      U(    ;
      U     "G271M".A_3125_MXZ01MA.Ma.StStartedFwd; // min one fan must run
      O     DB371.DBX 1445.2; // min one fan must run
      )     ;
      UN    "MAL1S032Par".Par.FlagProcess.Inf08; // Schritt halten
      UN    "G269M".A_3191_BTE07.OutOverflow; //LUFTTEMPERATUR ÜBER DER HORDE
      UN    "G269M".A_3191_BTE07.OutFaultAI; //LUFTTEMPERATUR ÜBER DER HORDE
      UN    "G269M".A_3191_BTE01.OutOverflow; //LUFTTEMPERATUR UNTER DER HORDE
      UN    "G269M".A_3191_BTE01.OutFaultAI; //LUFTTEMPERATUR UNTER DER HORDE
      SPBN  NoTi; // count steptime only when fan running and sensor alive
//JV161209      L     "MAL1S032Par".Par.ProcessValue.StepTimeAct    // in ms
//JV161209      L     #tmpCyclusTime
//JV161209      +D
//JV161209      T     "MAL1S032Par".Par.ProcessValue.StepTimeAct    // in ms
//--Create actual Timeinterval for counting steptime new JV151209 ===>

      CALL "SIEMENS_READ_CLK" (
           RET_VAL                  := MW   200,
           CDT                      := "MAL1S032Par".Par.ProcessValue.ActualTime);

      U     "MAL1S032Par".Par.FlagProcess.Inf04; // Zeitauswertung aktiv
      SPB   diff;
      CALL "SIEMENS_READ_CLK" (
           RET_VAL                  := MW   200,
           CDT                      := "MAL1S032Par".Par.ProcessValue.ActualTimePreviousScan);// Start-Zeit CPU-Clock aktuelle Auswertung
      SET   ;
      S     "MAL1S032Par".Par.FlagProcess.Inf04; // Zeitauswertung aktiv

diff: NOP   0;

      CALL "SB_DT_DT" (
           DT1                      := "MAL1S032Par".Par.ProcessValue.ActualTime,// momentane Zeit CPU-Clock
           DT2                      := "MAL1S032Par".Par.ProcessValue.ActualTimePreviousScan,// Start-Zeit CPU-Clock aktuelle Auswertung
           RET_VAL                  := "MAL1S032Par".Par.ProcessValue.Afeesttijd);// Zeitdifferenz in ms


      L     "MAL1S032Par".Par.ProcessValue.Afeesttijd; // Zeitdifferenz in ms
      L     L#10000; // 10sec
      >=D   ;
      R     "MAL1S032Par".Par.FlagProcess.Inf04; // Zeitauswertung aktiv
      FP    "MAL1S032Par".Par.FlagProcess.Inf05;
      SPBN  NoST;
      L     "MAL1S032Par".Par.ProcessValue.Afeesttijd; // Zeitdifferenz in ms
      SPM   Korr; //JV161209 Da hat wer an der Uhr gedreht.....
      L     L#10150; // 10sec + 150ms  als Maximalüberwachung
      >D    ; //JV161209 Da hat wer an der Uhr gedreht.....
      SPBN  AlOK;
Korr: NOP   0;
      L     L#10000; // 10sec als Grundwert, wenn die Zeit verstellt wurde
      T     "MAL1S032Par".Par.ProcessValue.Afeesttijd; // Zeitdifferenz in ms
AlOK: NOP   0;
      L     "MAL1S032Par".Par.ProcessValue.Afeesttijd; // Zeitdifferenz in ms
      L     "ASW_GraphicData".General.CycleTime[1].Actual; // aktuelle Zykluszeit als Korrektur
      +D    ;
      L     "MAL1S032Par".Par.ProcessValue.StepTimeAct; // in ms
      +D    ;
      T     "MAL1S032Par".Par.ProcessValue.StepTimeAct; // in ms
NoST: NOP   0;
//--Create actual Timeinterval for counting steptime new JV151209 <===

      SPA   OKTi; //JV161209
NoTi: NOP   0;
      SET   ; //JV161209 ===>
      R     "MAL1S032Par".Par.FlagProcess.Inf04; // Zeitauswertung aktiv
//JV161209 <===
OKTi: NOP   0; //JV161209
      L     "MAL1S032Par".Par.ProcessValue.StepTimeAct; // in ms
      L     L#86400000; // ms/d
      MOD   ;
      L     L#3600000; // ms/h
      /D    ;
      T     "MAL1S032Par".ActTimeStepProcess.SteptimeActHour; // Steptime in h

      L     "MAL1S032Par".Par.ProcessValue.StepTimeAct;
      L     L#3600000; // ms/h
      MOD   ;
      L     L#60000; // ms/min
      /D    ;
      T     "MAL1S032Par".ActTimeStepProcess.SteptimeActMin; // Steptime in min

      L     "MAL1S032Par".Par.ProcessValue.StepTimeAct;
      L     L#60000; // ms/min
      /D    ;
      T     "MAL1S032Par".ActTimeStepProcess.SteptimeActMinOverall; // Steptime in min overall

//
// Next Step
//
//   Switch over to next step under conditions:
//   or Maximal steptime
//   or Minimal steptime
//           and
//               or no setpoint delta temp
//               or atual value delta temp is ge setpoint deltatemp
//                   and sensor is ok
//           and
// /              or no setpoint max temp above floor
//              or atual value max temp above floor is ge setpoint max temp above floor
//                  and sensor is ok
// 1 Kriterium
      U(    ;
      L     "MAL1S032Par".ActTimeStepProcess.SteptimeActMinOverall; // Steptime in min overall
      L     "MAL1S032Par".StepAct.StepTime_Max; // Target steptime actual step
      >=I   ;
      )     ;
      O(    ;
// 2 Kriterium
      O(    ;
      U(    ;
      L     "MAL1S032Par".StepAct.DeltaTempSwitchpointStep;
      L     0;
//JV230310      >=D
      >D    ; //JV230310
      )     ;
// condition, if analogue input is not damaaged   //
      UN    "G269M".A_3191_BTE07.OutOverflow; //AIR TEMPERATURE ABOVE FLOOR
      UN    "G269M".A_3191_BTE07.OutFaultAI; //AIR TEMPERATURE ABOVE FLOOR
      UN    "G269M".A_3191_BTE01.OutOverflow; //AIR TEMPERATURE BELOW FLOOR
      UN    "G269M".A_3191_BTE01.OutFaultAI; //AIR TEMPERATURE BELOW FLOOR
      U(    ;
      L     "G269M".A_3191_BTE01.OutValueUnits; // act value temperature below floor
      L     "G269M".A_3191_BTE07.OutValueUnits; // act value temperature above floor
      -D    ; // delta temp actual
      L     L#10;
      /D    ;
      L     "MAL1S032Par".StepAct.DeltaTempSwitchpointStep;
      <D    ;
      )     ;
      )     ;
// 3 Kriterium
      O(    ;
      U(    ;
      L     "MAL1S032Par".StepAct.MaxTempAboveFloorStep;
      L     L#0; // 0,0°C is illegally switchpoint for max. temperature
      >D    ;
      )     ;
// condition, if analogue input is not damaaged   // MW R2.1
      UN    "G269M".A_3191_BTE01.OutOverflow; //AIR TEMPERATURE BELOW FLOOR
      UN    "G269M".A_3191_BTE01.OutFaultAI; //AIR TEMPERATURE BELOW FLOOR
      U(    ;
      L     "G269M".A_3191_BTE07.OutValueUnits; // act value temperature above floor
      L     L#10;
      /D    ;
      L     "MAL1S032Par".StepAct.MaxTempAboveFloorStep;
      >=D   ;
      )     ;
      )     ;
// 4 Kriterium
// and min. time
      U(    ;
      L     "MAL1S032Par".ActTimeStepProcess.SteptimeActMinOverall; // Steptime in min overall
      L     "MAL1S032Par".StepAct.StepTime_Min; // Target steptime actual step
      >=I   ;
      )     ;
      )     ;
// and not cooling                                // UK 22.01.07
      UN    "MAL1S032Par".Par.FlagProcess.Cooling_Activ;
// 5 Kriterium
      O(    ;
      U     "MAL1S032Par".Par.FlagProcess.Cooling_Activ;
      U(    ;
      L     "G269M".A_3191_BTE07.OutValueUnits; // act value temperature above floor
      L     L#10;
      /D    ;
      L     "MAL1S032Par".StepAct.TemperaturAboveFloor;
      <=D   ;
      )     ;
      O(    ;
      L     "MAL1S032Par".Par.ParIntMachine.ActualStep;
//JV210710      L     25                          // max. 24 Schritte
      L     27; // max. 26 Schritte   //JV210710
      >=I   ;
      )     ;
      )     ;
// and min. time
      U(    ;
      L     "MAL1S032Par".ActTimeStepProcess.SteptimeActMinOverall; // Steptime in min overall
      L     "MAL1S032Par".StepAct.StepTime_Min; // Target steptime actual step
      >=I   ;
      )     ;
      SPBN  E606;
// send average step data to PIC
      SET   ;
      S     "MAL1S032StepValues".SendData; // send average step data to PIC
// Next step
      L     "MAL1S032Par".Par.ParIntMachine.ActualStep;
      L     "MAL1S032Par".RecipeHeader.NumberOfSteps;
      >I    ;
      SPB   Pedk; // Last step is finished
//BRT20100901 ====> Schritt halten
      U     "MAL1S032Par".Par.FlagProcess.Inf08; // Schritt halten
      SPB   E606;
//BRT20100901 <====
//
      L     "MAL1S032Par".Par.ParIntMachine.ActualStep;
      L     1;
      +I    ;
      T     "MAL1S032Par".Par.ParIntMachine.ActualStep;
      L     0;
      T     "MAL1S032Par".ActTimeStepProcess.SteptimeActMinOverall; // Steptime in min Overall
      SPA   E606;
Pedk: NOP   0; // Process has finished
      SET   ;
      R     "MAL1S032Par".Par.FlagProcess.ProcessActive;
      R     "MAL1S032Par".Par.FlagProcess.Cooling_Activ;
      S     "MAL1S032Par".Par.FlagProcess.ProcessEnd;
//
      L     0; // clear step number
      T     "MAL1S032Par".Par.ParIntMachine.ActualStep;
      T     "MAL1S032Par".StepAct.StepNumber;
E606: NOP   0;
NETWORK
TITLE =ASW_6080: Active step kilning
//
      U     "MAL1S032Par".Par.FlagProcess.ProcessActive;
      SPBN  E608;
// copy stepnr for visu
      L     "MAL1S032Par".Par.ParIntMachine.ActualStep;
      T     "MAL1S032Par".Par.ParIntProcess.ActualStep;
//MW 2010.04.16
      U(    ;
      L     "MAL1S032Par".StepAct.StepTime_Min;
      L     0;
      ==I   ;
      )     ;
      U(    ;
      L     "MAL1S032Par".StepAct.StepTime_Max;
      L     0;
      ==I   ;
      )     ;
      SPB   Nklk;
// basic speed  fans
      L     "MAL1S032Par".StepAct.SpeedVentilatorBasic;
      T     "MAL1S032Par".Par.ParIntProcess.SpeedVentilatorBasic;
// basic position exhaust air flaps
      L     "MAL1S032Par".StepAct.PosExhaustAirFlapBasic; // setpoint from recipe
      L     10; // convert to 0.1%
      *I    ;
      T     "MAL1S032Par".Par.ParIntProcess.PosExhaustAirFlapBasic;
// basic position withering air channel flaps
      L     "MAL1S032Par".StepAct.PosWitheringAirFlapBasic; // setpoint from recipe
      L     10; // convert to 0.1%
      *I    ;
      T     "MAL1S032Par".Par.ParIntProcess.PosWitheringAirFlapBasic;
// basic position recycling air channel flaps
      L     "MAL1S032Par".StepAct.PosRecycleAirFlapBasic; // setpoint from recipe
      L     10; // convert to 0.1%
      *I    ;
      T     "MAL1S032Par".Par.ParIntProcess.PosRecycAirFlapBasic;
      T     "MAL1S032Par".Par.ProcessValue.Value17; // Sollwert Umluftklappen Verbund
//MW 2010.04.16
// basic position fresh air flaps
//      L     "MAL1S032Par".StepAct.PosFreshAirFlapBasic    // setpoint from recipe
      L     0; // 0%
      U     "MAL1S032Par".Par.FlagProcess.ProcessActive;
      UN    "MAL1S032Par".Par.FlagProcess.Cooling_Activ;
      SPB   klk;
      L     100; // 100%
      U     "MAL1S032Par".Par.FlagProcess.ProcessActive;
      U     "MAL1S032Par".Par.FlagProcess.Cooling_Activ;
      SPB   klk;
      SPA   Nklk;
klk:  L     10; // convert to 0.1%
      *I    ;
      T     "MAL1S032Par".Par.ParIntProcess.PosFreshAirFlapBasic;
Nklk: NOP   0;

// Nachlauf der Brenner
//    U     "GCS7_GrCtrlDB".OutEnable[276]    // G276M Heating Kilningbox
      U     "MAL1S032Par".Par.FlagProcess.ProcessActive;
      UN    "MAL1S032Par".Par.FlagProcess.Cooling_Activ;
      =     "MAL1S032Par".Par.FlagProcess.ProgrammSchwelkenDarren;

      U     "MAL1S032Par".Par.FlagProcess.ProgrammSchwelkenDarren;
      L     S5T#1M;
      SA    T     50; // Nachlauf Brenner

      UN    "MAL1S032Par".Par.FlagProcess.ProgrammSchwelkenDarren;
      U     T     50; // Nachlauf Brenner
      =     "MAL1S032Par".Par.FlagProcess1.HilfsRegler_1_Down;
      =     "MAL1S032Par".Par.FlagProcess1.HilfsRegler_2_Down;
      =     "MAL1S032Par".Par.FlagProcess1.HilfsRegler_3_Down;
      =     "MAL1S032Par".Par.FlagProcess1.HilfsRegler_4_Down;

// Sollwert - Istwert vergleich der Temperatur unter der Horde
      L     "MAL1S032Par".StepAct.TemperaturBelowFloor; // setpoint from SCADA
      L     L#10;
      *D    ;
      T     "MAL1S032Par".Par.ProcessValue.TemperaturBelowFloor;

      U     "SYS_Scan0_Tick1min";
      SPBN  NORM;
//- nur alle x Minuten korrigieren ---
      L     "MAL1S032Par".Par.ProcessValue.CorrInterval;
      +     1;
      T     "MAL1S032Par".Par.ProcessValue.CorrInterval;
      L     2; // Korrekturintervall [min]
      >=I   ;
      SPBN  NORM;
      L     0;
      T     "MAL1S032Par".Par.ProcessValue.CorrInterval;

      L     "MAL1S032Par".Par.ProcessValue.TemperaturBelowFloor;
      L     "G269M".A_3191_BTE01.OutValueUnits; // Real-Value Temperature below floor
      -D    ;
      L     50; // Totband in [0.5°C]
      <=D   ;
      SPB   uebe; // wenn größer keine Korrektur
//- zur Sicherheit nicht mehr als 5.0°C zulassen ---
      L     5.000000e+002; // max. Korrektur !
      L     "MAL1S032Par".Par.ProcessValue_Real.SollwertTempKorr;
      <=R   ;
      SPB   uebe;
      L     "MAL1S032Par".Par.ProcessValue_Real.SollwertTempKorr;
      L     1.000000e+000; // Anpassung an Differenz zwischen den PT100
      +R    ;
      T     "MAL1S032Par".Par.ProcessValue_Real.SollwertTempKorr;
uebe: NOP   0;

      L     "MAL1S032Par".Par.ProcessValue.TemperaturBelowFloor;
      L     "G269M".A_3191_BTE01.OutValueUnits; // Real-Value Temperature below floor
      -D    ;
      L     50; // Totband in [0.5°C]
      >=D   ;
      SPB   unte; // wenn kleier keine Korrektur
//- keine negative Korrektur (führt sonst zu Schwingung) ---
      L     0.000000e+000; // keine negative Korrektur !
      L     "MAL1S032Par".Par.ProcessValue_Real.SollwertTempKorr;
      >=R   ;
      SPB   unte;
      L     1.000000e+000; // Anpassung an Differenz zwischen den PT100
      -R    ;
      T     "MAL1S032Par".Par.ProcessValue_Real.SollwertTempKorr;
unte: NOP   0;

//- bei Schrittbegin noch keine Korrektur ---
NORM: L     "MAL1S032Par".ActTimeStepProcess.SteptimeActMinOverall; // Steptime in min overall
      L     8; // Korrekturverzögerung [min]
      >I    ;
      SPB   SET;
      L     0.000000e+000;
      T     "MAL1S032Par".Par.ProcessValue_Real.SollwertTempKorr;
      L     10; // grossen Wert in Intervallzähler vorladen ...
      T     "MAL1S032Par".Par.ProcessValue.CorrInterval; // ... damit nächster 1MinTick gleich wirksam wird

SET:  NOP   0;
      L     "MAL1S032Par".Par.ProcessValue.TemperaturBelowFloor;
      DTR   ;
      L     "MAL1S032Par".Par.ProcessValue_Real.SollwertTempKorr;
      +R    ;
      T     "MAL1S032Par".Par.ProcessValue_Real.T_SOLL_NORM;
      SPA   M641;
      NOP   0;
//- Korrekturfaktor auf "0" setzen ---
      L     0.000000e+000;
      T     "MAL1S032Par".Par.ProcessValue_Real.SollwertTempKorr;
M641: NOP   0;
      SPA   GCPR;

// GCPRO
// setpoint temperature below floor
      NOP   0; // setpoint fans automatic mode
      L     L#0;
      U     "MAL1S032Par".Par.FlagProcess.Cooling_Activ; // switch over to cooling
      SPB   aut1;
      L     "MAL1S032Par".StepAct.TemperaturBelowFloor; // setpoint from SCADA
aut1: NOP   0;
      DTR   ;
      L     1.000000e+001;
      /R    ;
      T     "MAL1S032Par".Par.ProcessValue_Real.T_SOLL_NORM;
// emergency kiln heating
// fan 1
      U(    ;
      L     2#1;
      L     "MAL1S032Par".RecipeHeader.DeselectVentilator; // emergency regime without fan 1
      ==I   ;
      )     ;
      L     "G269M".A_3191_BTE05.OutValuePc; //AIR TEMPERATURE DIFFUSOR FAN 1 :  temperature in diffusor fan 1
      SPBN  c1R1;
      L     "G269M".A_3191_BTE01.OutValuePc; //AIR TEMPERATURE BELOW FLOOR
      L     "G269M".A_3191_BTE05.OutValuePc; //AIR TEMPERATURE DIFFUSOR FAN 1 :  temperature in diffusor fan 2
      <D    ;
      SPBN  c1R1;
      TAK   ;
c1R1: T     "MAL1S032Par".Par.ParIntProcess.ActValueTemperature_R1;
// fan 2
      U(    ;
      L     2#10;
      L     "MAL1S032Par".RecipeHeader.DeselectVentilator; // emergency regime without fan 2
      ==I   ;
      )     ;
      L     "G269M".A_3191_BTE05.OutValuePc; //AIR TEMPERATURE DIFFUSOR FAN 1 :  temperature in diffusor fan 2
      SPBN  c1R2;
      L     "G269M".A_3191_BTE01.OutValuePc; //AIR TEMPERATURE BELOW FLOOR
      L     "G269M".A_3191_BTE05.OutValuePc; //AIR TEMPERATURE DIFFUSOR FAN 1 :  temperature in diffusor fan 1
      <D    ;
      SPBN  c1R2;
      TAK   ;
c1R2: T     "MAL1S032Par".Par.ParIntProcess.ActValueTemperature_R2;

GCPR: NOP   0;
//BRT20100901 ====> Schritt halten, wenn in Rezept aktiviert!!!
      U(    ;
      L     "MAL1S032Par".RecipeHeader.SPARE_DINT004;
      L     L#1; // Schritt halten aktiviert = 1
      ==D   ;
      )     ;
      U(    ;
      L     "G269M".A_3191_BTE07.OutValuePc; // Temperature above floor kiln 2
      L     100;
      /D    ;
      L     "MAL1S032Par".RecipeHeader.SPARE_INT002; // Schaltpunkt für Schritt halten
      >=I   ;
      )     ;
      U(    ;
      U     "MAL1S033".ToASW.InfDataReady; // Kiln 1 bereit
      O     "MAL1S033Par".Par.FlagFunction_1.StepLoading;
      )     ;
      UN    "MAL1S033Par".Par.FlagProcess.ProcessActive;
      UN(   ;
      U     "G297M".A_3225_MXZ01MA.Ma.StStartedFwd;
      U     "G297M".A_3225_TSC01_AF.OutL; // Ventilator 1 dreht mind. 40% SW
      U     "G297M".A_3226_MXZ01MA.Ma.StStartedFwd;
      U     "G297M".A_3226_TSC01_AF.OutL; // Ventilator 2 dreht mind. 40% SW
      )     ;
      S     "MAL1S032Par".Par.FlagProcess.Inf08; // Schritt halten

      U(    ;
      L     "MAL1S032Par".RecipeHeader.SPARE_DINT004;
      L     L#1; // Schritt halten aktiviert = 1
      <>D   ;
      )     ;
      O(    ;
      U     "MAL1S033Par".Par.FlagProcess.ProcessActive;
      U(    ;
      U     "G297M".A_3225_MXZ01MA.Ma.StStartedFwd;
      U     "G297M".A_3225_TSC01_AF.OutL; // Ventilator 1 dreht mind. 40% SW
      O     ;
      U     "G297M".A_3226_MXZ01MA.Ma.StStartedFwd;
      U     "G297M".A_3226_TSC01_AF.OutL; // Ventilator 2 dreht mind. 40% SW
      )     ;
      )     ;
      R     "MAL1S032Par".Par.FlagProcess.Inf08; // Schritt halten
//BRT20100901 <====
// cooling down
      L     "MAL1S032Par".StepAct.CoolingDown;
      L     1;
      ==I   ;
      S     "MAL1S032Par".Par.FlagProcess.Cooling_Activ;
//JV250710 =====>
      L     "MAL1S032Par".Par.ParIntMachine.ActualStep;
      L     24;
      <I    ;
      O(    ; //JV290710 ======>
      L     "MAL1S032Par".StepAct.CoolingDown;
      L     1;
      <>I   ;
      )     ; //JV290710 <=====
      R     "MAL1S032Par".Par.FlagProcess.Cooling_Activ;
//JV250710 <=====
E608: NOP   0;
//BRT20100901 ====> Schritt-Halte-Bit wird nochmals explizit bei Prozess Ende zurückgesetzt!!!
      UN    "MAL1S032Par".Par.FlagProcess.ProcessActive;
      O     "MAL1S032Par".Par.FlagProcess.ProcessEnd;
      R     "MAL1S032Par".Par.FlagProcess.Inf08; // Schritt halten


// Abdarr-Betrieb aktiv
      U(    ;
      L     "MAL1S032Par".Par.ParIntMachine.ActualStep;
      L     "MAL1S033Par".Par.ParIntMachine.ActualStep;
      >I    ;
      )     ;
      UN    "MAL1S032Par".Par.FlagProcess.Cooling_Activ;
      O     "MAL1S033Par".Par.FlagProcess.Cooling_Activ;
//BRT20100830 ====> Bit Abdarr Betrieb Aktiv abhängig von Rezeptwert!
//      =     "MAL1S032Par".Par.FlagProcess.Abdarr_Betrieb_Aktiv
      =     "MAL1S032Par".Par.FlagProcess2.Inf22; // Hilfsbit für Abdarr-Betrieb

      U     "MAL1S032Par".Par.FlagProcess2.Inf22; // Hilfsbit für Abdarr-Betrieb
      U(    ; // Schaltpunkt Schwelken/Darren aus Line Parameter
      L     "G269M".A_3191_BTE07.OutValuePc; // Temperature above floor
      L     L#100;
      /D    ;
//      L     "MAL1Par".Values1.Value04   // Line Parameter
      L     "MAL1S032Par".RecipeHeader.SPARE_INT000; // Rezept Parameter
      >=D   ;
      )     ;
      S     "MAL1S032Par".Par.FlagProcess.Abdarr_Betrieb_Aktiv;

      UN    "MAL1S032Par".Par.FlagProcess2.Inf22; // Hilfsbit für Abdarr-Betrieb
      R     "MAL1S032Par".Par.FlagProcess.Abdarr_Betrieb_Aktiv;
//BRT20100830 <====

//BRT20100830 ====> Regelung während Verbundbetrieb!!!
//
      U     "MAL1S032Par".Par.FlagProcess.ProcessActive;
      U     "MAL1S032Par".Par.FlagProcess.Abdarr_Betrieb_Aktiv;
      U(    ;
      L     "MAL1S032Par".Par.ParIntMachine.ActualStep;
      L     "MAL1S032Par".Par.ProcessValue.Value16; // Step-Copy
      >I    ;
      )     ;
      FP    "MAL1S032Par".Par.FlagProcess2.Inf23;
      =     "MAL1S032Par".Par.FlagProcess2.Inf24;

//Einlesen der Rezeptwerte jeden neuen Schritt!
      U     "MAL1S032Par".Par.FlagProcess2.Inf24;
      O(    ;
      L     "MAL1S032Par".RecipeHeader.SPARE_DINT0003;
      L     L#1; // autom. Regelung ON = 1
      <>D   ;
      )     ;
      ON(   ;
      L     "G269M".A_3191_BTE07.OutValuePc; // Temperature above floor kiln 1
      L     5500; // 55°C
      >=I   ;
      )     ;
      SPBN  rd01;
      L     "MAL1S032Par".Par.ParIntMachine.ActualStep;
      T     "MAL1S032Par".Par.ProcessValue.Value16; // Step-Copy

      L     "MAL1S032Par".Par.ParIntProcess.PosRecycAirFlapBasic; // setpoint from recipe
      T     "MAL1S032Par".Par.ProcessValue.Value17; // Sollwert Umluftklappen Verbund

      L     "MAL1S032Par".Par.ParIntProcess.SpeedVentilatorBasic; // setpoint from recipe
      T     "MAL1S032Par".Par.ProcessValue.Value18; // Sollwert Ventilator Verbund
rd01: NOP   0;

//BRT20100903 ====> Verzögerung nach Step-Wechsel bis Regelung aktiv!
      U     "MAL1S032Par".Par.FlagProcess2.Inf24;
      L     S5T#15M;
      SV    T     30;
//BRT20100903 <====

      U     "MAL1S032Par".Par.FlagProcess.ProcessActive;
      U     "MAL1S032Par".Par.FlagProcess.Abdarr_Betrieb_Aktiv;
      U(    ;
      L     "MAL1S032Par".RecipeHeader.SPARE_DINT0003;
      L     L#1; // autom. Regelung ON = 1
      ==D   ;
      )     ;
      UN    T     30; // Verzögerung nach Step-Wechsel   //BRT20100903
      UN    T     31; // alle 5 min kann geregelt werden
      U(    ;
      L     "G269M".A_3191_BTE07.OutValuePc; // Temperature above floor kiln 1
      L     5500; // 55°C
      >=I   ;
      )     ;
      SPBN  nore;
      L     "MAL1S033Par".StepAct.TemperaturBelowFloor;
      L     10;
      -I    ;
      L     10;
      *I    ;
      L     "G295M".A_3291_BTE01.OutValuePc; // Temperature below floor kiln 2
      >I    ;
      SPB   pls1;
      L     "MAL1S033Par".StepAct.TemperaturBelowFloor;
      L     10;
      +I    ;
      L     10;
      *I    ;
      L     "G295M".A_3291_BTE01.OutValuePc; // Temperature below floor kiln 2
      <I    ;
      SPB   mns1;
      SPA   recl;
pls1: NOP   0;
//      L     "MAL1S032Par".Par.ProcessValue.Value17    // Sollwert Umluftklappen Verbund
//      L     50                          // 5%
//      -D
//      T     "MAL1S032Par".Par.ProcessValue.Value17    // Sollwert Umluftklappen Verbund

      L     "MAL1S032Par".Par.ProcessValue.Value18; // Sollwert Ventilator Verbund
      L     L#2; // 2%
      +D    ;
      T     "MAL1S032Par".Par.ProcessValue.Value18; // Sollwert Ventilator Verbund
      SPA   recl;
mns1: NOP   0;
//      L     "MAL1S032Par".Par.ProcessValue.Value17    // Sollwert Umluftklappen Verbund
//      L     50                          // 5%
//      +D
//      T     "MAL1S032Par".Par.ProcessValue.Value17    // Sollwert Umluftklappen Verbund

      L     "MAL1S032Par".Par.ProcessValue.Value18; // Sollwert Ventilator Verbund
      L     L#2; // 2%
      -D    ;
      T     "MAL1S032Par".Par.ProcessValue.Value18; // Sollwert Ventilator Verbund
recl: NOP   0;

//Kontrolle der Regelwerte Umluftklappen Grenzwerte Min/Max
//      L     "MAL1S032Par".Par.ProcessValue.Value17    // Sollwert Umluftklappen Verbund
//      L     "MAL1S032Par".Par.ParIntProcess.PosRecycAirFlapBasic    // setpoint from recipe
//      <D
//      SPB   min1
//      TAK
//min1: T     "MAL1S032Par".Par.ProcessValue.Value17    // Sollwert Umluftklappen Verbund

//      L     "MAL1S032Par".Par.ProcessValue.Value17    // Sollwert Umluftklappen Verbund
//      L     L#900                       // maximum 90%
//      >D
//      SPB   max1
//      TAK
//max1: T     "MAL1S032Par".Par.ProcessValue.Value17    // Sollwert Umluftklappen Verbund

//Kontrolle der Regelwerte Ventilator Grenzwerte Min/max
      L     "MAL1S032Par".Par.ProcessValue.Value18; // Sollwert Ventilator Verbund
      L     L#60; // minimum 60%
      <D    ;
      SPB   min2;
      TAK   ;
min2: T     "MAL1S032Par".Par.ProcessValue.Value18; // Sollwert Ventilator Verbund

      L     "MAL1S032Par".Par.ProcessValue.Value18; // Sollwert Ventilator Verbund
      L     L#100; // maximum 100%
      >D    ;
      SPB   max2;
      TAK   ;
max2: T     "MAL1S032Par".Par.ProcessValue.Value18; // Sollwert Ventilator Verbund
nore: NOP   0;

// 5 min Tick für Regelung
      UN    T     31;
      L     S5T#5M;
      SV    T     31;

//BRT20100830 <====

//BRT20100826 ====> neu mit geregelter Abkühlung!
//
      U     "MAL1S032Par".Par.FlagProcess.Cooling_Activ;
      FP    "MAL1S032Par".Par.FlagProcess2.Inf20;
      =     "MAL1S032Par".Par.FlagProcess2.Inf21;

      U     "MAL1S032Par".Par.FlagProcess2.Inf21;
      O(    ; // in Schritt 25/26 nach Rezeptwert fahren !!!
      L     "MAL1S032Par".Par.ParIntMachine.ActualStep;
      L     24;
      >I    ;
      )     ;
      SPBN  read;
      L     "MAL1S032Par".StepAct.MaxTempAboveFloorStep;
      T     "MAL1S032Par".Par.ProcessValue.Value13; // Schaltpunkt Regelung

      L     "MAL1S032Par".Par.ParIntProcess.PosRecycAirFlapBasic; // setpoint from recipe
      T     "MAL1S032Par".Par.ProcessValue.Value14; // Sollwert Umluftklappen Kühlen

      L     "MAL1S032Par".Par.ParIntProcess.SpeedVentilatorBasic; // setpoint from recipe
      T     "MAL1S032Par".Par.ProcessValue.Value15; // Sollwert Ventilator Kühlen
read: NOP   0;


      L     "G269M".A_3191_BTE07.OutValuePc; // Temperature above floor
      L     L#10;
      /D    ;
      L     "MAL1S032Par".Par.ProcessValue.Value13; // Schaltpunkt Regelung
      <D    ;
      U(    ; // Regelung nur im Schritt 24 !!!
      L     "MAL1S032Par".Par.ParIntMachine.ActualStep;
      L     24;
      ==I   ;
      )     ;
      U     "SYS_Scan0_Tick30s"; // zur Sicherheit
      SPBN  cont;
//neuen Schaltpunkt für nächsten Schritt generieren
      L     "MAL1S032Par".Par.ProcessValue.Value13; // Schaltpunkt Regelung
      L     L#20; // 2,0° C
      -D    ;
      T     "MAL1S032Par".Par.ProcessValue.Value13; // Schaltpunkt Regelung

      L     "MAL1S032Par".Par.ProcessValue.Value14; // Sollwert Umluftklappen Kühlen
      L     L#100; // 10%
      -D    ;
      L     L#0; // Überwachung min. Position
      <=D   ;
      SPB   null;
      TAK   ;
null: T     "MAL1S032Par".Par.ProcessValue.Value14; // Sollwert Umluftklappen Kühlen


      L     "MAL1S032Par".Par.ProcessValue.Value15; // Sollwert Ventilator Kühlen
      L     L#6; // 6%
      +D    ;
      L     L#100; // Überwachung max. Drehzahl
      >=D   ;
      SPB   hdrt;
      TAK   ;
hdrt: T     "MAL1S032Par".Par.ProcessValue.Value15; // Sollwert Ventilator Kühlen

cont: NOP   0;
NETWORK
TITLE =ASW_6090: calculate heat quantity active kilning

      L     L#0;
      U     "MAL1S032Par".Par.FlagProcess.ProcessActive;
      SPBN  n609; // no addition
      SET   ;
      S     "MAL1S032Par".Par.FlagProcess.Inf21; // add heat quantity
      U     "SYS_Scan0_Tick1s"; // scan 1sec
      SPBN  E609;
      L     "MAL1S032Par".Par.ProcessValue_Real.Value05; // heat quantity in kW
      +R    ;
      T     "MAL1S032Par".Par.ProcessValue_Real.Value05;
      SPA   E609;
n609: NOP   0;
      U     "MAL1S032Par".Par.FlagProcess.Inf21; // add heat quantity
      SPBN  E609;
      R     "MAL1S032Par".Par.FlagProcess.Inf21; // add heat quantity
      L     "MAL1S032Par".Par.ProcessValue_Real.Value05;
      L     3.600000e+003;
      /R    ; // from kWs to kWh
      L     1.000000e+003;
      /R    ; // from kWh to MWh
      RND   ;
      T     "MAL1S032Par".Par.ProcessValue_Real.Value06; // result to batch potokoll
      L     0.000000e+000; // clear calculator
      T     "MAL1S032Par".Par.ProcessValue_Real.Value05;
E609: NOP   0;
NETWORK
TITLE =ASW_7000: Step loading kilning
//       U     "MAL1S032".ToASW.InfDataReady
//      U     "MAL1S032".PCRead.Step.StWait
//      U     "MAL1S032".PCWrite.ExtFuncOn.StartLoading    // PIC command "start
//loading"
//      S     "MAL1S032Par".Par.FlagFunction_1.StepLoading    // Step loading
//      R     "MAL1S032Par".Par.FlagMachine.ImpulsNullstellung
//      R     "MAL1S032Par".Par.FlagMachine.CmdTurnRevAfterLoading
//      R     "MAL1S032Par".Par.FlagMachine.CmdTurnFwdAfterLoading
////
//      SET
//      R     "MAL1S032".PCWrite.ExtFuncOn.StartLoading    // PIC command "start
//loading"
////
//      U     "MAL1S032".ToASW.InfDataReady
//      U     "MAL1S032".PCRead.Step.StActive
//      U     "MAL1S032Par".Par.FlagFunction_1.StepLoading    // Step loading
//      SPB   e71
//      R     "MAL1S032Par".Par.Switches1.StaOn00    // LiftingPositionRound_1
//      R     "MAL1S032Par".Par.Switches1.StaOn01    // LiftingPositionRound_2
//      R     "MAL1S032Par".Par.Switches1.StaOn02    // LiftingPositionRound_3
//      R     "MAL1S032Par".Par.Switches1.StaOn03    // LiftingPositionRound_4
//      R     "MAL1S032Par".Par.Switches1.StaOn04    // LiftingPositionRound_5
//      R     "MAL1S032Par".Par.Switches1.StaOn05    // LiftingPositionRound_6
//e71:  NOP   0
//      U     "MAL1S032".ToASW.InfDataReady
//      U     "MAL1S032".PCRead.Step.StActive
//      U     "MAL1S032Par".Par.FlagFunction_1.StepLoading    // Step loading
//      UN    "MAL1S032Par".Par.FlagFunction_1.FinishLoading
//      UN    "MAL1S032Par".Par.FlagFunction_1.LoadEnd
//      SPBN  E700
//      U(
//      U(
//      L     "G266M".A_3111_MXZ41MA.Ma.OutPositionAngle
//      L     3460                        // 346.0°
//      >=I
//      )
//      O
//      U(
//      L     "G266M".A_3111_MXZ41MA.Ma.OutCntRound
//      L     L#1
//      >=D
//      )
//      )
//      U     "MAL1S032Par".Par.FlagFunction_1.StepLoading
//      =     "MAL1S032Par".Par.FlagFunction_0.ReducedSpeed
////
//      L     "MAL1S032Par".RecipeHeader.Loading.LiftingPositionRound_3
//      L     20                          // 20°
//      -I
//      T     "MAL1S032Par".Par.ParIntMachine.LiftingPositionRound_4
//      L     "MAL1S032Par".RecipeHeader.Loading.LoadingLevelRound_3
//      L     "MAL1S032Par".RecipeHeader.Loading.OffsetLevelNextRound
//      +I
//      T     "MAL1S032Par".Par.ParIntMachine.LoadingLevelRound_4
////
//      L     "MAL1S032Par".Par.ParIntMachine.LiftingPositionRound_4
//      L     20                          // 20°
//      -I
//      T     "MAL1S032Par".Par.ParIntMachine.LiftingPositionRound_5
//      L     "MAL1S032Par".Par.ParIntMachine.LoadingLevelRound_4
//      L     "MAL1S032Par".RecipeHeader.Loading.OffsetLevelNextRound
//      +I
//      T     "MAL1S032Par".Par.ParIntMachine.LoadingLevelRound_5
////
//      L     "MAL1S032Par".Par.ParIntMachine.LiftingPositionRound_5
//      L     20                          // 20°
//      -I
//      T     "MAL1S032Par".Par.ParIntMachine.LiftingPositionRound_6
//      L     "MAL1S032Par".Par.ParIntMachine.LoadingLevelRound_5
//      L     "MAL1S032Par".RecipeHeader.Loading.OffsetLevelNextRound
//      +I
//      T     "MAL1S032Par".Par.ParIntMachine.LoadingLevelRound_6
////
//      L     3600
//      L     "G266M".A_3111_MXZ41MA.Ma.Par.ParTolPosition
//      -I
//      L     "G266M".A_3111_MXZ41MA.Ma.OutPositionAngle
//      <=I
//      SPB   E700
////
//      L     "G266M".A_3111_MXZ41MA.Ma.OutPositionAngle
//      L     0
//      <I
////      <=I
//      SPB   E700
////
//      L     "G266M".A_3111_MXZ41MA.Ma.OutPositionAngle
//      L     10
//      /I
//      T     "MAL1S032Par".Par.MachineValue.ISTWERT_FAHRANTRIEB_POSI
////
//      U     "MAL1S032Par".Par.FlagFunction_1.StepLoading    // Step loading
//      FP    "MAL1S032Par".Par.Switches1.StaOn08
//      =     "MAL1S032Par".Par.Switches1.StaOn09    // scan start loading
//      U     "MAL1S032Par".Par.Switches1.StaOn09    // scan start loading
//      SPBN  e72
//      R     "MAL1S032Par".Par.Switches1.StaOn00    // LiftingPositionRound_1
//      R     "MAL1S032Par".Par.Switches1.StaOn01    // LiftingPositionRound_2
//      R     "MAL1S032Par".Par.Switches1.StaOn02    // LiftingPositionRound_3
//      R     "MAL1S032Par".Par.Switches1.StaOn03    // LiftingPositionRound_4
//      R     "MAL1S032Par".Par.Switches1.StaOn04    // LiftingPositionRound_5
//      R     "MAL1S032Par".Par.Switches1.StaOn05    // LiftingPositionRound_6
////
//e72:  NOP   0
////
//      U(
//      L     "G266M".A_3111_MXZ41MA.Ma.OutCntRound
//      L     L#0
//      ==D
//      )
//      U(
//      L     "MAL1S032Par".Par.MachineValue.ISTWERT_FAHRANTRIEB_POSI
//      L     "MAL1S032Par".RecipeHeader.Loading.LiftingPositionRound_1
//      <I
//      )
//      S     "MAL1S032Par".Par.Switches1.StaOn00    // LiftingPositionRound_1
////
//      U(
//      L     "G266M".A_3111_MXZ41MA.Ma.OutCntRound
//      L     L#0
//      ==D
//      )
//      U(
//      L     "MAL1S032Par".Par.MachineValue.ISTWERT_FAHRANTRIEB_POSI
//      L     "MAL1S032Par".RecipeHeader.Loading.LiftingPositionRound_1
//      >=I
//      )
//      U(
//      L     "MAL1S032Par".Par.MachineValue.ISTWERT_FAHRANTRIEB_POSI
//      L     3550                        // 355.0° --> Ruckeln am Nullpunkt
//abfangen
//      <=I
//      )
//      S     "MAL1S032Par".Par.Switches1.StaOn01    // LiftingPositionRound_2
////
//      U     "MAL1S032Par".Par.Switches1.StaOn01    // LiftingPositionRound_2
//      R     "MAL1S032Par".Par.Switches1.StaOn00    // LiftingPositionRound_1
////
//      U(
//      L     "G266M".A_3111_MXZ41MA.Ma.OutCntRound
//      L     L#1
//      ==D
//      )
//      U(
//      L     "MAL1S032Par".Par.MachineValue.ISTWERT_FAHRANTRIEB_POSI
//      L     "MAL1S032Par".RecipeHeader.Loading.LiftingPositionRound_2
//      >=I
//      )
//      S     "MAL1S032Par".Par.Switches1.StaOn02    // LiftingPositionRound_3
////
//      U     "MAL1S032Par".Par.Switches1.StaOn02    // LiftingPositionRound_3
//      R     "MAL1S032Par".Par.Switches1.StaOn01    // LiftingPositionRound_2
//      R     "MAL1S032Par".Par.Switches1.StaOn00    // LiftingPositionRound_1
////
//      U(
//      L     "G266M".A_3111_MXZ41MA.Ma.OutCntRound
//      L     L#2
//      ==D
//      )
//      U(
//      L     "MAL1S032Par".Par.MachineValue.ISTWERT_FAHRANTRIEB_POSI
//      L     "MAL1S032Par".RecipeHeader.Loading.LiftingPositionRound_3
//      >=I
//      )
//      S     "MAL1S032Par".Par.Switches1.StaOn03    // LiftingPositionRound_4
////
//      U     "MAL1S032Par".Par.Switches1.StaOn03    // LiftingPositionRound_4
//      R     "MAL1S032Par".Par.Switches1.StaOn02    // LiftingPositionRound_3
//      R     "MAL1S032Par".Par.Switches1.StaOn01    // LiftingPositionRound_2
//      R     "MAL1S032Par".Par.Switches1.StaOn00    // LiftingPositionRound_1
//      U(
//      L     "G266M".A_3111_MXZ41MA.Ma.OutCntRound
//      L     L#3
//      ==D
//      )
//      U(
//      L     "MAL1S032Par".Par.MachineValue.ISTWERT_FAHRANTRIEB_POSI
//      L     "MAL1S032Par".Par.ParIntMachine.LiftingPositionRound_4
//      >=I
//      )
//      S     "MAL1S032Par".Par.Switches1.StaOn04    // LiftingPositionRound_5
////
//      U     "MAL1S032Par".Par.Switches1.StaOn04    // LiftingPositionRound_5
//      R     "MAL1S032Par".Par.Switches1.StaOn03    // LiftingPositionRound_4
//      R     "MAL1S032Par".Par.Switches1.StaOn02    // LiftingPositionRound_3
//      R     "MAL1S032Par".Par.Switches1.StaOn01    // LiftingPositionRound_2
//      R     "MAL1S032Par".Par.Switches1.StaOn00    // LiftingPositionRound_1
//      U(
//      L     "G266M".A_3111_MXZ41MA.Ma.OutCntRound
//      L     L#4
//      ==D
//      )
//      U(
//      L     "MAL1S032Par".Par.MachineValue.ISTWERT_FAHRANTRIEB_POSI
//      L     "MAL1S032Par".Par.ParIntMachine.LiftingPositionRound_5
//      >=I
//      )
//      S     "MAL1S032Par".Par.Switches1.StaOn05    // LiftingPositionRound_6
////
//      U     "MAL1S032Par".Par.Switches1.StaOn05    // LiftingPositionRound_6
//      R     "MAL1S032Par".Par.Switches1.StaOn04    // LiftingPositionRound_5
//      R     "MAL1S032Par".Par.Switches1.StaOn03    // LiftingPositionRound_4
//      R     "MAL1S032Par".Par.Switches1.StaOn02    // LiftingPositionRound_3
//      R     "MAL1S032Par".Par.Switches1.StaOn01    // LiftingPositionRound_2
//      R     "MAL1S032Par".Par.Switches1.StaOn00    // LiftingPositionRound_1
//      U     "MAL1S032Par".Par.Switches1.StaOn00    // LiftingPositionRound_1
//      SPB   Rnd1
//      U     "MAL1S032Par".Par.Switches1.StaOn01    // LiftingPositionRound_2
//      SPB   Rnd2
//      U     "MAL1S032Par".Par.Switches1.StaOn02    // LiftingPositionRound_3
//      SPB   Rnd3
//      U     "MAL1S032Par".Par.Switches1.StaOn03    // LiftingPositionRound_4
//      SPB   Rnd4
//      U     "MAL1S032Par".Par.Switches1.StaOn04    // LiftingPositionRound_5
//      SPB   Rnd5
//      U     "MAL1S032Par".Par.Switches1.StaOn05    // LiftingPositionRound_6
//      SPB   Rnd6
//      SPA   E700
//Rnd1: NOP   0
//      L     "MAL1S032Par".RecipeHeader.Loading.LoadingLevelRound_1
//      L     "G265M".A_3111_MXZ21_31MA.Ma.Par.ParTolPosition
//      +I
//      T     "MAL1S032Par".Par.MachineValue.SOLLWERT_HUBZUG1_HOEHE
//      T     "MAL1S032Par".Par.MachineValue.SOLLWERT_HUBZUG2_HOEHE
//      L     "MAL1S032Par".RecipeHeader.Loading.LoadingSpeed_1
//      T     "MAL1S032Par".Par.MachineValue.SollwertFahrantrieb
//      SPA   E700
//Rnd2: NOP   0
//      L     "MAL1S032Par".RecipeHeader.Loading.LoadingLevelRound_2
//      L     "G265M".A_3111_MXZ21_31MA.Ma.Par.ParTolPosition
//      +I
//      T     "MAL1S032Par".Par.MachineValue.SOLLWERT_HUBZUG1_HOEHE
//      T     "MAL1S032Par".Par.MachineValue.SOLLWERT_HUBZUG2_HOEHE
//      L     "MAL1S032Par".RecipeHeader.Loading.LoadingSpeed_2
//      T     "MAL1S032Par".Par.MachineValue.SollwertFahrantrieb
//      SPA   E700
//Rnd3: NOP   0
//      L     "MAL1S032Par".RecipeHeader.Loading.LoadingLevelRound_3
//      L     "G265M".A_3111_MXZ21_31MA.Ma.Par.ParTolPosition
//      +I
//      T     "MAL1S032Par".Par.MachineValue.SOLLWERT_HUBZUG1_HOEHE
//      T     "MAL1S032Par".Par.MachineValue.SOLLWERT_HUBZUG2_HOEHE
//      L     "MAL1S032Par".RecipeHeader.Loading.LoadingSpeed_3
//      T     "MAL1S032Par".Par.MachineValue.SollwertFahrantrieb
//      SPA   E700
//Rnd4: NOP   0
//      L     "MAL1S032Par".Par.ParIntMachine.LoadingLevelRound_4
//      L     "G265M".A_3111_MXZ21_31MA.Ma.Par.ParTolPosition
//      +I
//      T     "MAL1S032Par".Par.MachineValue.SOLLWERT_HUBZUG1_HOEHE
//      T     "MAL1S032Par".Par.MachineValue.SOLLWERT_HUBZUG2_HOEHE
////      L     "MAL1S032Par".RecipeHeader.Loading.LoadingSpeed_3
//      L     87                          // 87%
//      T     "MAL1S032Par".Par.MachineValue.SollwertFahrantrieb
//      SPA   E700
//Rnd5: NOP   0
//      L     "MAL1S032Par".Par.ParIntMachine.LoadingLevelRound_5
//      L     "G265M".A_3111_MXZ21_31MA.Ma.Par.ParTolPosition
//      +I
//      T     "MAL1S032Par".Par.MachineValue.SOLLWERT_HUBZUG1_HOEHE
//      T     "MAL1S032Par".Par.MachineValue.SOLLWERT_HUBZUG2_HOEHE
////      L     "MAL1S032Par".RecipeHeader.Loading.LoadingSpeed_3
//      L     87                          // 87%
//      T     "MAL1S032Par".Par.MachineValue.SollwertFahrantrieb
//      SPA   E700
//Rnd6: NOP   0
//      L     "MAL1S032Par".Par.ParIntMachine.LoadingLevelRound_6
//      L     "G265M".A_3111_MXZ21_31MA.Ma.Par.ParTolPosition
//      +I
//      T     "MAL1S032Par".Par.MachineValue.SOLLWERT_HUBZUG1_HOEHE
//      T     "MAL1S032Par".Par.MachineValue.SOLLWERT_HUBZUG2_HOEHE
////      L     "MAL1S032Par".RecipeHeader.Loading.LoadingSpeed_3
//      L     87                          // 87%
//      T     "MAL1S032Par".Par.MachineValue.SollwertFahrantrieb
//      SPA   E700
//E700: NOP   0
//
      U     "MAL1S032".ToASW.InfDataReady;
      U     "MAL1S032".PCRead.Step.StWait;
      U     "MAL1S032".PCWrite.ExtFuncOn.StartLoading; // PIC command "start loading"
      S     "MAL1S032Par".Par.FlagFunction_1.StepLoading; // Step loading
      R     "MAL1S032Par".Par.FlagMachine.ImpulsNullstellung;
      R     "MAL1S032Par".Par.FlagMachine.CmdTurnRevAfterLoading;
      R     "MAL1S032Par".Par.FlagMachine.CmdTurnFwdAfterLoading;
//MW 2010.04.06
      R     "MAL1S032Par".Par.FlagFunction_0.MerkerBeladenGestartetFP;
//
      SET   ;
      R     "MAL1S032".PCWrite.ExtFuncOn.StartLoading; // PIC command "start loading"
//
//MW 2010.04.06
      U     "MAL1S032Par".Par.FlagFunction_1.StepLoading;
      U     "MAL1S032".ToASW.InfSameBatchPrevSec;
      S     "MAL1S032Par".Par.FlagFunction_0.MerkerBeladenGestartetFP;
//
      U     "MAL1S032".ToASW.InfDataReady;
      U     "MAL1S032".PCRead.Step.StActive;
      U     "MAL1S032Par".Par.FlagFunction_1.StepLoading; // Step loading
      SPB   e71;
      R     "MAL1S032Par".Par.Switches1.StaOn00; // LiftingPositionRound_1
      R     "MAL1S032Par".Par.Switches1.StaOn01; // LiftingPositionRound_2
      R     "MAL1S032Par".Par.Switches1.StaOn02; // LiftingPositionRound_3
      R     "MAL1S032Par".Par.Switches1.StaOn03; // LiftingPositionRound_4
      R     "MAL1S032Par".Par.Switches1.StaOn04; // LiftingPositionRound_5
      R     "MAL1S032Par".Par.Switches1.StaOn05; // LiftingPositionRound_6
e71:  NOP   0;
//
      U     "MAL1S032".ToASW.InfDataReady;
      U     "MAL1S032".PCRead.Step.StActive;
      U     "MAL1S032Par".Par.FlagFunction_1.StepLoading; // Step loading
//MW 2010.04.06      UN    "MAL1S032Par".Par.FlagFunction_1.FinishLoading
//MW 2010.04.06      UN    "MAL1S032Par".Par.FlagFunction_1.LoadEnd
      SPBN  E700;
      U(    ;
      U(    ;
      L     "G266M".A_3111_MXZ41MA.Ma.OutPositionAngle;
      L     3460; // 346.0°
      >=I   ;
      )     ;
      O     ;
      U(    ;
      L     "G266M".A_3111_MXZ41MA.Ma.OutCntRound;
      L     L#1;
      >=D   ;
      )     ;
      )     ;
      U     "MAL1S032Par".Par.FlagFunction_1.StepLoading;
      =     "MAL1S032Par".Par.FlagFunction_0.ReducedSpeed;
//
      L     "MAL1S032Par".RecipeHeader.Loading.LiftingPositionRound_3;
      L     20; // 20°
      -I    ;
      T     "MAL1S032Par".Par.ParIntMachine.LiftingPositionRound_4;
      L     "MAL1S032Par".RecipeHeader.Loading.LoadingLevelRound_3;
      L     "MAL1S032Par".RecipeHeader.Loading.OffsetLevelNextRound;
      +I    ;
      T     "MAL1S032Par".Par.ParIntMachine.LoadingLevelRound_4;
//
      L     "MAL1S032Par".Par.ParIntMachine.LiftingPositionRound_4;
      L     20; // 20°
      -I    ;
      T     "MAL1S032Par".Par.ParIntMachine.LiftingPositionRound_5;
      L     "MAL1S032Par".Par.ParIntMachine.LoadingLevelRound_4;
      L     "MAL1S032Par".RecipeHeader.Loading.OffsetLevelNextRound;
      +I    ;
      T     "MAL1S032Par".Par.ParIntMachine.LoadingLevelRound_5;
//
      L     "MAL1S032Par".Par.ParIntMachine.LiftingPositionRound_5;
      L     20; // 20°
      -I    ;
      T     "MAL1S032Par".Par.ParIntMachine.LiftingPositionRound_6;
      L     "MAL1S032Par".Par.ParIntMachine.LoadingLevelRound_5;
      L     "MAL1S032Par".RecipeHeader.Loading.OffsetLevelNextRound;
      +I    ;
      T     "MAL1S032Par".Par.ParIntMachine.LoadingLevelRound_6;
//
      L     3600;
      L     "G266M".A_3111_MXZ41MA.Ma.Par.ParTolPosition;
      -I    ;
      L     "G266M".A_3111_MXZ41MA.Ma.OutPositionAngle;
      <=I   ;
      SPB   E700;
//MW 2010.04.06
      L     3600;
      L     "G266M".A_3111_MXZ41MA.Ma.Par.ParTolPosition;
      -I    ;
      L     "G266M".A_3111_MXZ41MA.Ma.OutPositionAngle;
      <=I   ;
      U     "G266M".A_3111_MXZ41MA.A_3111_MXZ41.OutpRunFwd;
      SPB   E700;
//
//MW 2010.04.06      L     "G266M".A_3111_MXZ41MA.Ma.OutPositionAngle
//MW 2010.04.06      L     0
//MW 2010.04.06      <I
//MW 2010.04.06//      <=I
//MW 2010.04.06
      L     "G266M".A_3111_MXZ41MA.Ma.OutPositionAngle;
      L     0;
      <=I   ;
      U     "G266M".A_3111_MXZ41MA.A_3111_MXZ41.OutpRunFwd;
      SPB   E700;
//
      L     "G266M".A_3111_MXZ41MA.Ma.OutPositionAngle;
      L     10;
      /I    ;
      T     "MAL1S032Par".Par.MachineValue.ISTWERT_FAHRANTRIEB_POSI;
//
      U     "MAL1S032Par".Par.FlagFunction_1.StepLoading; // Step loading
      FP    "MAL1S032Par".Par.Switches1.StaOn08;
      =     "MAL1S032Par".Par.Switches1.StaOn09; // scan start loading
      U     "MAL1S032Par".Par.Switches1.StaOn09; // scan start loading
      SPBN  e72;
      R     "MAL1S032Par".Par.Switches1.StaOn00; // LiftingPositionRound_1
      R     "MAL1S032Par".Par.Switches1.StaOn01; // LiftingPositionRound_2
      R     "MAL1S032Par".Par.Switches1.StaOn02; // LiftingPositionRound_3
      R     "MAL1S032Par".Par.Switches1.StaOn03; // LiftingPositionRound_4
      R     "MAL1S032Par".Par.Switches1.StaOn04; // LiftingPositionRound_5
      R     "MAL1S032Par".Par.Switches1.StaOn05; // LiftingPositionRound_6
//
e72:  NOP   0;
//
      U(    ;
      L     "G266M".A_3111_MXZ41MA.Ma.OutCntRound;
      L     L#0;
      ==D   ;
      )     ;
      U(    ;
      L     "MAL1S032Par".Par.MachineValue.ISTWERT_FAHRANTRIEB_POSI;
      L     "MAL1S032Par".RecipeHeader.Loading.LiftingPositionRound_1;
      <I    ;
      )     ;
      S     "MAL1S032Par".Par.Switches1.StaOn00; // LiftingPositionRound_1
//
      U(    ;
      L     "G266M".A_3111_MXZ41MA.Ma.OutCntRound;
      L     L#0;
      ==D   ;
      )     ;
      U(    ;
      L     "MAL1S032Par".Par.MachineValue.ISTWERT_FAHRANTRIEB_POSI;
      L     "MAL1S032Par".RecipeHeader.Loading.LiftingPositionRound_1;
      >=I   ;
      )     ;
      U(    ;
      L     "MAL1S032Par".Par.MachineValue.ISTWERT_FAHRANTRIEB_POSI;
      L     3550; // 355.0° --> Ruckeln am Nullpunkt abfangen
      <=I   ;
      )     ;
      S     "MAL1S032Par".Par.Switches1.StaOn01; // LiftingPositionRound_2
//
      U     "MAL1S032Par".Par.Switches1.StaOn01; // LiftingPositionRound_2
      R     "MAL1S032Par".Par.Switches1.StaOn00; // LiftingPositionRound_1
//
      U(    ;
      L     "G266M".A_3111_MXZ41MA.Ma.OutCntRound;
      L     L#1;
      ==D   ;
      )     ;
      U(    ;
      L     "MAL1S032Par".Par.MachineValue.ISTWERT_FAHRANTRIEB_POSI;
      L     "MAL1S032Par".RecipeHeader.Loading.LiftingPositionRound_2;
      >=I   ;
      )     ;
//MW 2010.04.06
      U(    ;
      L     "MAL1S032Par".Par.MachineValue.ISTWERT_FAHRANTRIEB_POSI;
      L     "MAL1S032Par".RecipeHeader.Loading.LiftingPositionRound_1;
      <I    ;
      )     ;
      S     "MAL1S032Par".Par.Switches1.StaOn02; // LiftingPositionRound_3
//
      U     "MAL1S032Par".Par.Switches1.StaOn02; // LiftingPositionRound_3
      R     "MAL1S032Par".Par.Switches1.StaOn01; // LiftingPositionRound_2
      R     "MAL1S032Par".Par.Switches1.StaOn00; // LiftingPositionRound_1
//
      U(    ;
      L     "G266M".A_3111_MXZ41MA.Ma.OutCntRound;
      L     L#2;
      ==D   ;
      )     ;
      U(    ;
      L     "MAL1S032Par".Par.MachineValue.ISTWERT_FAHRANTRIEB_POSI;
      L     "MAL1S032Par".RecipeHeader.Loading.LiftingPositionRound_3;
      >=I   ;
      )     ;
//MW 2010.04.06
      U(    ;
      L     "MAL1S032Par".Par.MachineValue.ISTWERT_FAHRANTRIEB_POSI;
      L     "MAL1S032Par".RecipeHeader.Loading.LiftingPositionRound_2;
      <I    ;
      )     ;
      S     "MAL1S032Par".Par.Switches1.StaOn03; // LiftingPositionRound_4
//
      U     "MAL1S032Par".Par.Switches1.StaOn03; // LiftingPositionRound_4
      R     "MAL1S032Par".Par.Switches1.StaOn02; // LiftingPositionRound_3
      R     "MAL1S032Par".Par.Switches1.StaOn01; // LiftingPositionRound_2
      R     "MAL1S032Par".Par.Switches1.StaOn00; // LiftingPositionRound_1
      U(    ;
      L     "G266M".A_3111_MXZ41MA.Ma.OutCntRound;
      L     L#3;
      ==D   ;
      )     ;
      U(    ;
      L     "MAL1S032Par".Par.MachineValue.ISTWERT_FAHRANTRIEB_POSI;
      L     "MAL1S032Par".Par.ParIntMachine.LiftingPositionRound_4;
      >=I   ;
      )     ;
//MW 2010.04.06
      U(    ;
      L     "MAL1S032Par".Par.MachineValue.ISTWERT_FAHRANTRIEB_POSI;
      L     "MAL1S032Par".RecipeHeader.Loading.LiftingPositionRound_3;
      <I    ;
      )     ;
      S     "MAL1S032Par".Par.Switches1.StaOn04; // LiftingPositionRound_5
//
      U     "MAL1S032Par".Par.Switches1.StaOn04; // LiftingPositionRound_5
      R     "MAL1S032Par".Par.Switches1.StaOn03; // LiftingPositionRound_4
      R     "MAL1S032Par".Par.Switches1.StaOn02; // LiftingPositionRound_3
      R     "MAL1S032Par".Par.Switches1.StaOn01; // LiftingPositionRound_2
      R     "MAL1S032Par".Par.Switches1.StaOn00; // LiftingPositionRound_1
      U(    ;
      L     "G266M".A_3111_MXZ41MA.Ma.OutCntRound;
      L     L#4;
      ==D   ;
      )     ;
      U(    ;
      L     "MAL1S032Par".Par.MachineValue.ISTWERT_FAHRANTRIEB_POSI;
      L     "MAL1S032Par".Par.ParIntMachine.LiftingPositionRound_5;
      >=I   ;
      )     ;
//MW 2010.04.06
      U(    ;
      L     "MAL1S032Par".Par.MachineValue.ISTWERT_FAHRANTRIEB_POSI;
      L     "MAL1S032Par".RecipeHeader.Loading.LiftingPositionRound_4;
      <I    ;
      )     ;
      S     "MAL1S032Par".Par.Switches1.StaOn05; // LiftingPositionRound_6
//
      U     "MAL1S032Par".Par.Switches1.StaOn05; // LiftingPositionRound_6
      R     "MAL1S032Par".Par.Switches1.StaOn04; // LiftingPositionRound_5
      R     "MAL1S032Par".Par.Switches1.StaOn03; // LiftingPositionRound_4
      R     "MAL1S032Par".Par.Switches1.StaOn02; // LiftingPositionRound_3
      R     "MAL1S032Par".Par.Switches1.StaOn01; // LiftingPositionRound_2
      R     "MAL1S032Par".Par.Switches1.StaOn00; // LiftingPositionRound_1
      U     "MAL1S032Par".Par.Switches1.StaOn00; // LiftingPositionRound_1
      SPB   Rnd1;
      U     "MAL1S032Par".Par.Switches1.StaOn01; // LiftingPositionRound_2
      SPB   Rnd2;
      U     "MAL1S032Par".Par.Switches1.StaOn02; // LiftingPositionRound_3
      SPB   Rnd3;
      U     "MAL1S032Par".Par.Switches1.StaOn03; // LiftingPositionRound_4
      SPB   Rnd4;
      U     "MAL1S032Par".Par.Switches1.StaOn04; // LiftingPositionRound_5
      SPB   Rnd5;
      U     "MAL1S032Par".Par.Switches1.StaOn05; // LiftingPositionRound_6
      SPB   Rnd6;
      SPA   E700;
Rnd1: NOP   0;
      L     "MAL1S032Par".RecipeHeader.Loading.LoadingLevelRound_1;
      L     "G265M".A_3111_MXZ21_31MA.Ma.Par.ParTolPosition;
      +I    ;
      T     "MAL1S032Par".Par.MachineValue.SOLLWERT_HUBZUG1_HOEHE;
      T     "MAL1S032Par".Par.MachineValue.SOLLWERT_HUBZUG2_HOEHE;
      L     "MAL1S032Par".RecipeHeader.Loading.LoadingSpeed_1;
      T     "MAL1S032Par".Par.MachineValue.SollwertFahrantrieb;
      SPA   E700;
Rnd2: NOP   0;
      L     "MAL1S032Par".RecipeHeader.Loading.LoadingLevelRound_2;
      L     "G265M".A_3111_MXZ21_31MA.Ma.Par.ParTolPosition;
      +I    ;
      T     "MAL1S032Par".Par.MachineValue.SOLLWERT_HUBZUG1_HOEHE;
      T     "MAL1S032Par".Par.MachineValue.SOLLWERT_HUBZUG2_HOEHE;
      L     "MAL1S032Par".RecipeHeader.Loading.LoadingSpeed_2;
      T     "MAL1S032Par".Par.MachineValue.SollwertFahrantrieb;
      SPA   E700;
Rnd3: NOP   0;
      L     "MAL1S032Par".RecipeHeader.Loading.LoadingLevelRound_3;
      L     "G265M".A_3111_MXZ21_31MA.Ma.Par.ParTolPosition;
      +I    ;
      T     "MAL1S032Par".Par.MachineValue.SOLLWERT_HUBZUG1_HOEHE;
      T     "MAL1S032Par".Par.MachineValue.SOLLWERT_HUBZUG2_HOEHE;
      L     "MAL1S032Par".RecipeHeader.Loading.LoadingSpeed_3;
      T     "MAL1S032Par".Par.MachineValue.SollwertFahrantrieb;
      SPA   E700;
Rnd4: NOP   0;
      L     "MAL1S032Par".Par.ParIntMachine.LoadingLevelRound_4;
      L     "G265M".A_3111_MXZ21_31MA.Ma.Par.ParTolPosition;
      +I    ;
      T     "MAL1S032Par".Par.MachineValue.SOLLWERT_HUBZUG1_HOEHE;
      T     "MAL1S032Par".Par.MachineValue.SOLLWERT_HUBZUG2_HOEHE;
//      L     "MAL1S032Par".RecipeHeader.Loading.LoadingSpeed_3
      L     87; // 87%
      T     "MAL1S032Par".Par.MachineValue.SollwertFahrantrieb;
      SPA   E700;
Rnd5: NOP   0;
      L     "MAL1S032Par".Par.ParIntMachine.LoadingLevelRound_5;
      L     "G265M".A_3111_MXZ21_31MA.Ma.Par.ParTolPosition;
      +I    ;
      T     "MAL1S032Par".Par.MachineValue.SOLLWERT_HUBZUG1_HOEHE;
      T     "MAL1S032Par".Par.MachineValue.SOLLWERT_HUBZUG2_HOEHE;
//      L     "MAL1S032Par".RecipeHeader.Loading.LoadingSpeed_3
      L     87; // 87%
      T     "MAL1S032Par".Par.MachineValue.SollwertFahrantrieb;
      SPA   E700;
Rnd6: NOP   0;
      L     "MAL1S032Par".Par.ParIntMachine.LoadingLevelRound_6;
      L     "G265M".A_3111_MXZ21_31MA.Ma.Par.ParTolPosition;
      +I    ;
      T     "MAL1S032Par".Par.MachineValue.SOLLWERT_HUBZUG1_HOEHE;
      T     "MAL1S032Par".Par.MachineValue.SOLLWERT_HUBZUG2_HOEHE;
//      L     "MAL1S032Par".RecipeHeader.Loading.LoadingSpeed_3
      L     87; // 87%
      T     "MAL1S032Par".Par.MachineValue.SollwertFahrantrieb;
      SPA   E700;
E700: NOP   0;
NETWORK
TITLE =Sub 7010: Kilning  loading finished
//// Grundschicht vollständig bedeckt
//      U(
//// Die Position bei IBN ermitteln!
//      L     "G266M".A_3111_MXZ41MA.Ma.OutPositionAngle
//      L     3564                        // 356.4°
//      >=I
//      )
//      U     "MAL1S032Par".Par.FlagFunction_1.StepLoading
//      U     "G266M".A_3111_MXZ41MA.Ma.InEnableFwd
//      S     "MAL1S032Par".Par.FlagFunction_1.LoadFirstPartEnd
//      S     "MAL1S032Par".Par.FlagProcess.Product_Inside
//
//      U     "MAL1S032Par".Par.FlagProcess.ProcessActive
//      U     "MAL1S032Par".Par.FlagFunction_1.FinishLoading
//      O     "MAL1S032Par".Par.FlagFunction_1.StepUnloading
//      O     "MAL1S032".PCRead.Step.StIdling    // "SecDB".PCRead.Step.StIdling
//      R     "MAL1S032Par".Par.FlagFunction_1.LoadFirstPartEnd
//
//      L     0
//      L     "MAL1S032".ToSSW.InPrevSecDB
//      ==I
//      SPB   fin
//      O(
////KR10022010      U     "MAL1S017Par".Par.FlagFunction_1.FinishUnloading
////KR10022010      U     "MAL1S017".PCWrite.ExtFuncOn.FinishCleanSurface    //
//PIC command "finish unloading"
//      U     "MAL1S032".PCWrite.ExtFuncOn.FinishLoading    // PIC command
//"finish
//loading"
//      O     "MAL1S017Par".Par.FlagFunction_1.StepCleaning
////KR10022010      U     "MAL1S017".PCRead.Step.StEmptied
//      U(
//      AUF   "MAL1S017"
//      L     DBNO
//      L     "MAL1S032".ToSSW.InPrevSecDB
//      ==I
//      )
//      )
//      O(
//      U     "MAL1S018Par".Par.FlagFunction_1.FinishUnloading
//      U     "MAL1S018".PCWrite.ExtFuncOn.FinishCleanSurface    // PIC command
//"finish unloading"
////      U     "MAL1S032".PCWrite.ExtFuncOn.FinishLoading    // PIC command
//"finish loading"
//      O     "MAL1S018Par".Par.FlagFunction_1.StepCleaning
//      U     "MAL1S018".PCRead.Step.StEmptied
//      U(
//      AUF   "MAL1S018"
//      L     DBNO
//      L     "MAL1S032".ToSSW.InPrevSecDB
//      ==I
//      )
//      )
//      O(
//      U     "MAL1S019Par".Par.FlagFunction_1.FinishUnloading
//      U     "MAL1S019".PCWrite.ExtFuncOn.FinishCleanSurface    // PIC command
//"finish unloading"
////      U     "MAL1S032".PCWrite.ExtFuncOn.FinishLoading    // PIC command
//"finish loading"
//      O     "MAL1S019Par".Par.FlagFunction_1.StepCleaning
//      U     "MAL1S019".PCRead.Step.StEmptied
//      U(
//      AUF   "MAL1S019"
//      L     DBNO
//      L     "MAL1S032".ToSSW.InPrevSecDB
//      ==I
//      )
//      )
//      O(
//      U     "MAL1S020Par".Par.FlagFunction_1.FinishUnloading
//      U     "MAL1S020".PCWrite.ExtFuncOn.FinishCleanSurface    // PIC command
//"finish unloading"
////      U     "MAL1S032".PCWrite.ExtFuncOn.FinishLoading    // PIC command
//"finish loading"
//      O     "MAL1S020Par".Par.FlagFunction_1.StepCleaning
//      U     "MAL1S020".PCRead.Step.StEmptied
//      U(
//      AUF   "MAL1S020"
//      L     DBNO
//      L     "MAL1S032".ToSSW.InPrevSecDB
//      ==I
//      )
//      )
//      O(
//      U     "MAL1S021Par".Par.FlagFunction_1.FinishUnloading
//      U     "MAL1S021".PCWrite.ExtFuncOn.FinishCleanSurface    // PIC command
//"finish unloading"
////      U     "MAL1S032".PCWrite.ExtFuncOn.FinishLoading    // PIC command
//"finish loading"
//      O     "MAL1S021Par".Par.FlagFunction_1.StepCleaning
//      U     "MAL1S021".PCRead.Step.StEmptied
//      U(
//      AUF   "MAL1S021"
//      L     DBNO
//      L     "MAL1S032".ToSSW.InPrevSecDB
//      ==I
//      )
//      )
//      O(
//      U     "MAL1S022Par".Par.FlagFunction_1.FinishUnloading
//      U     "MAL1S022".PCWrite.ExtFuncOn.FinishCleanSurface    // PIC command
//"finish unloading"
////      U     "MAL1S032".PCWrite.ExtFuncOn.FinishLoading    // PIC command
//"finish loading"
//      O     "MAL1S022Par".Par.FlagFunction_1.StepCleaning
//      U     "MAL1S022".PCRead.Step.StEmptied
//      U(
//      AUF   "MAL1S022"
//      L     DBNO
//      L     "MAL1S032".ToSSW.InPrevSecDB
//      ==I
//      )
//      )
//      O(
//      U     "MAL1S023Par".Par.FlagFunction_1.FinishUnloading
//      U     "MAL1S023".PCWrite.ExtFuncOn.FinishCleanSurface    // PIC command
//"finish unloading"
////      U     "MAL1S032".PCWrite.ExtFuncOn.FinishLoading    // PIC command
//"finish loading"
//      O     "MAL1S032Par".Par.FlagFunction_1.StepCleaning
//      U     "MAL1S032".PCRead.Step.StEmptied
//      U(
//      AUF   "MAL1S023"
//      L     DBNO
//      L     "MAL1S023".ToSSW.InPrevSecDB
//      ==I
//      )
//      )
//      O(
//      U     "MAL1S024Par".Par.FlagFunction_1.FinishUnloading
//      U     "MAL1S024".PCWrite.ExtFuncOn.FinishCleanSurface    // PIC command
//"finish unloading"
////      U     "MAL1S032".PCWrite.ExtFuncOn.FinishLoading    // PIC command
//"finish loading"
//      O     "MAL1S024Par".Par.FlagFunction_1.StepCleaning
//      U     "MAL1S024".PCRead.Step.StEmptied
//      U(
//      AUF   "MAL1S024"
//      L     DBNO
//      L     "MAL1S032".ToSSW.InPrevSecDB
//      ==I
//      )
//      )
////      O(
////      U     "MAL1S032Par".Par.FlagFunction_1.StepLoading    // Step loading
////      UN    "MAL1S032".ToASW.InfSameJobPrevSec
////      U     "MAL1S032".PCWrite.ExtFuncOn.FinishLoading    // PIC command
//"finish loading"
////      )
//      U     "MAL1S032".ToASW.InfDataReady
//      U     "MAL1S032".PCRead.Step.StActive
//      U     "MAL1S032Par".Par.FlagFunction_1.LoadFirstPartEnd
//      S     "MAL1S032Par".Par.FlagFunction_1.LoadEnd
//      R     "MAL1S017".PCWrite.ExtFuncOn.FinishCleanSurface    // PIC command
//"finish unloading"
//      R     "MAL1S018".PCWrite.ExtFuncOn.FinishCleanSurface    // PIC command
//"finish unloading"
//      R     "MAL1S019".PCWrite.ExtFuncOn.FinishCleanSurface    // PIC command
//"finish unloading"
//      R     "MAL1S020".PCWrite.ExtFuncOn.FinishCleanSurface    // PIC command
//"finish unloading"
//      R     "MAL1S021".PCWrite.ExtFuncOn.FinishCleanSurface    // PIC command
//"finish unloading"
//      R     "MAL1S022".PCWrite.ExtFuncOn.FinishCleanSurface    // PIC command
//"finish unloading"
//      R     "MAL1S023".PCWrite.ExtFuncOn.FinishCleanSurface    // PIC command
//"finish unloading"
//      R     "MAL1S024".PCWrite.ExtFuncOn.FinishCleanSurface    // PIC command
//"finish unloading"
//
////
//      U     "MAL1S032".PCWrite.ExtFuncOn.FinishLoading    // PIC command
//"finish
//loading"
//      R     "MAL1S032".PCWrite.ExtFuncOn.FinishLoading    // PIC command
//"finish
//loading"
////
//      U     "MAL1S032Par".Par.FlagFunction_1.LoadEnd
//      U     "MAL1S032Par".Par.FlagFunction_1.StepLoading    // Step loading
//      FP    "MAL1S032Par".Par.FlagFunction_0.ImpulsSollposition
//      =     "MAL1S032Par".Par.FlagFunction_0.MerkerSollpositionFP
//      U     "MAL1S032Par".Par.FlagFunction_0.MerkerSollpositionFP
//      SPBN  fin
//      L     "G266M".A_3111_MXZ41MA.Ma.OutPositionAngle
//      L     "MAL1S032Par".Par.ParIntProcess.LoadingOverlap
//      +I
//      T     "G266M".A_3111_MXZ41MA.Ma.InPositionTarget
//      SET
//      S     "G266M".TurningTo_Parkposition
//
//// Extra Planierrunde wenn der Fahrantrieb ueber 346° beim Beladen Ende war
//      L     "G266M".A_3111_MXZ41MA.Ma.OutPositionAngle
//      L     3460                        // 346,0 °
//      >I
//      S     "G266M".Turning_One_Round_More
//
//// Beladehöhe speichern
//      L     "MAL1S032Par".Par.MachineValue.SOLLWERT_HUBZUG1_HOEHE
//      T     "MAL1S032Par".Par.ParIntMachine.LastLoadingLevel    // saved
//loading
//value
//fin:  NOP   0
//
//// Hubzüge erst auf der Parkposition abheben
//      U     "G266M".TurningTo_Parkposition
//      FN    "G265M".USW8
//      =     "G265M".USW9
//
//      U     "G265M".USW9
//      O
//      U     "MAL1S032Par".Par.FlagFunction_1.FinishLoading
//      U(
//      U     "G266M".A_3111_MXZ41MA.A_3111_BZS43.StCtoTrue    // sensor zero
//point
//      O     "G266M".A_3111_MXZ41MA.A_3111_BZS43.StTrue    // sensor zero point
//      )
//      SPBN  auf
//      L     "G265M".A_3111_MXZ21_31MA.Ma.Par.ParPositionTopLeftUnits
////LIFTING DRIVE
//      L     150
//      +I
//      T     "MAL1S032Par".Par.MachineValue.SOLLWERT_HUBZUG1_HOEHE
//      L     "G265M".A_3111_MXZ21_31MA.Ma.Par.ParPositionTopRightUnits
////LIFTING DRIVE
//      L     150
//      +I
//      T     "MAL1S032Par".Par.MachineValue.SOLLWERT_HUBZUG2_HOEHE
//      L     1
//      T     "G265M".A_3111_MXZ21_31MA.Ma.Par.ParTolPosition
//auf:  NOP   0
//
//      NOP   0
//
// Grundschicht vollständig bedeckt
//MW 2010.04.06
      U(    ;
      L     "G266M".A_3111_MXZ41MA.Ma.OutPositionAngle;
      L     3580; // 358.0°
      <I    ;
      )     ;
      U(    ;
// Die Position bei IBN ermitteln!
      L     "G266M".A_3111_MXZ41MA.Ma.OutPositionAngle;
//MW 2010.04.06      L     3564                        // 356.4°
      L     3540; // 354.0°
      >=I   ;
      )     ;
      U     "MAL1S032Par".Par.FlagFunction_1.StepLoading;
      U     "G266M".A_3111_MXZ41MA.Ma.InEnableFwd;
      S     "MAL1S032Par".Par.FlagFunction_1.LoadFirstPartEnd;
      S     "MAL1S032Par".Par.FlagProcess.Product_Inside;

      U     "MAL1S032Par".Par.FlagProcess.ProcessActive;
      U     "MAL1S032Par".Par.FlagFunction_1.FinishLoading;
      O     "MAL1S032Par".Par.FlagFunction_1.StepUnloading;
      O     "MAL1S032".PCRead.Step.StIdling; // "SecDB".PCRead.Step.StIdling
      R     "MAL1S032Par".Par.FlagFunction_1.LoadFirstPartEnd;

      L     0;
      L     "MAL1S032".ToSSW.InPrevSecDB;
      ==I   ;
//MW 2010.04.06      SPB   fin
//MW 2010.04.06
      SPB   suki;
      O(    ;
      U     "MAL1S017Par".Par.FlagFunction_1.FinishUnloading;
      O     "MAL1S017Par".Par.FlagFunction_1.StepCleaning; // Step cleaning
      O     "MAL1S017Par".Par.FlagFunction_1.FinishCleaning;
      U     "MAL1S017".PCRead.Step.StEmptied;
      ON    "MAL1S017".ToASW.InfDataReady; //JV070810
      U     "MAL1S032".PCWrite.ExtFuncOn.FinishLoading; // PIC command "finish loading"
      U(    ;
      AUF   "MAL1S017";
      L     DBNO;
      L     "MAL1S032".ToSSW.InPrevSecDB;
      ==I   ;
      )     ;
      )     ;
      O(    ;
      U     "MAL1S018Par".Par.FlagFunction_1.FinishUnloading;
      O     "MAL1S018Par".Par.FlagFunction_1.StepCleaning; // Step cleaning
      O     "MAL1S018Par".Par.FlagFunction_1.FinishCleaning;
      U     "MAL1S018".PCRead.Step.StEmptied;
      ON    "MAL1S018".ToASW.InfDataReady; //JV070810
      U     "MAL1S032".PCWrite.ExtFuncOn.FinishLoading; // PIC command "finish loading"
      U(    ;
      AUF   "MAL1S018";
      L     DBNO;
      L     "MAL1S032".ToSSW.InPrevSecDB;
      ==I   ;
      )     ;
      )     ;
      O(    ;
      U     "MAL1S019Par".Par.FlagFunction_1.FinishUnloading;
      O     "MAL1S019Par".Par.FlagFunction_1.StepCleaning; // Step cleaning
      O     "MAL1S019Par".Par.FlagFunction_1.FinishCleaning;
      U     "MAL1S019".PCRead.Step.StEmptied;
      ON    "MAL1S019".ToASW.InfDataReady; //JV070810
      U     "MAL1S032".PCWrite.ExtFuncOn.FinishLoading; // PIC command "finish loading"
      U(    ;
      AUF   "MAL1S019";
      L     DBNO;
      L     "MAL1S032".ToSSW.InPrevSecDB;
      ==I   ;
      )     ;
      )     ;
      O(    ;
      U     "MAL1S020Par".Par.FlagFunction_1.FinishUnloading;
      O     "MAL1S020Par".Par.FlagFunction_1.StepCleaning; // Step cleaning
      O     "MAL1S020Par".Par.FlagFunction_1.FinishCleaning;
      U     "MAL1S020".PCRead.Step.StEmptied;
      ON    "MAL1S020".ToASW.InfDataReady; //JV070810
      U     "MAL1S032".PCWrite.ExtFuncOn.FinishLoading; // PIC command "finish loading"
      U(    ;
      AUF   "MAL1S020";
      L     DBNO;
      L     "MAL1S032".ToSSW.InPrevSecDB;
      ==I   ;
      )     ;
      )     ;
      O(    ;
      U     "MAL1S021Par".Par.FlagFunction_1.FinishUnloading;
      O     "MAL1S021Par".Par.FlagFunction_1.StepCleaning; // Step cleaning
      O     "MAL1S021Par".Par.FlagFunction_1.FinishCleaning;
      U     "MAL1S021".PCRead.Step.StEmptied;
      ON    "MAL1S021".ToASW.InfDataReady; //JV070810
      U     "MAL1S032".PCWrite.ExtFuncOn.FinishLoading; // PIC command "finish loading"
      U(    ;
      AUF   "MAL1S021";
      L     DBNO;
      L     "MAL1S032".ToSSW.InPrevSecDB;
      ==I   ;
      )     ;
      )     ;
      O(    ;
      U     "MAL1S022Par".Par.FlagFunction_1.FinishUnloading;
      O     "MAL1S022Par".Par.FlagFunction_1.StepCleaning; // Step cleaning
      O     "MAL1S022Par".Par.FlagFunction_1.FinishCleaning;
      U     "MAL1S022".PCRead.Step.StEmptied;
      ON    "MAL1S022".ToASW.InfDataReady; //JV070810
      U     "MAL1S032".PCWrite.ExtFuncOn.FinishLoading; // PIC command "finish loading"
      U(    ;
      AUF   "MAL1S022";
      L     DBNO;
      L     "MAL1S032".ToSSW.InPrevSecDB;
      ==I   ;
      )     ;
      )     ;
      O(    ;
      U     "MAL1S023Par".Par.FlagFunction_1.FinishUnloading;
      O     "MAL1S023Par".Par.FlagFunction_1.StepCleaning; // Step cleaning
      O     "MAL1S023Par".Par.FlagFunction_1.FinishCleaning;
      U     "MAL1S023".PCRead.Step.StEmptied;
      ON    "MAL1S023".ToASW.InfDataReady; //JV070810
      U     "MAL1S032".PCWrite.ExtFuncOn.FinishLoading; // PIC command "finish loading"
      U(    ;
      AUF   "MAL1S023";
      L     DBNO;
      L     "MAL1S032".ToSSW.InPrevSecDB;
      ==I   ;
      )     ;
      )     ;
      O(    ;
      U     "MAL1S024Par".Par.FlagFunction_1.FinishUnloading;
      O     "MAL1S024Par".Par.FlagFunction_1.StepCleaning; // Step cleaning
      O     "MAL1S024Par".Par.FlagFunction_1.FinishCleaning;
      U     "MAL1S024".PCRead.Step.StEmptied;
      ON    "MAL1S024".ToASW.InfDataReady; //JV070810
      U     "MAL1S032".PCWrite.ExtFuncOn.FinishLoading; // PIC command "finish loading"
      U(    ;
      AUF   "MAL1S024";
      L     DBNO;
      L     "MAL1S032".ToSSW.InPrevSecDB;
      ==I   ;
      )     ;
      )     ;
suki: NOP   0;
      O(    ;
      U     "MAL1S032Par".Par.FlagFunction_1.StepLoading; // Step loading
      UN    "MAL1S032".ToASW.InfSameJobPrevSec;
      U     "MAL1S032".PCWrite.ExtFuncOn.FinishLoading; // PIC command "finish loading"
      )     ;
      U     "MAL1S032".ToASW.InfDataReady;
      U     "MAL1S032".PCRead.Step.StActive;
      U     "MAL1S032Par".Par.FlagFunction_1.LoadFirstPartEnd;
      S     "MAL1S032Par".Par.FlagFunction_1.LoadEnd;
      R     "MAL1S017".PCWrite.ExtFuncOn.FinishCleanSurface; // PIC command "finish unloading"
      R     "MAL1S018".PCWrite.ExtFuncOn.FinishCleanSurface; // PIC command "finish unloading"
      R     "MAL1S019".PCWrite.ExtFuncOn.FinishCleanSurface; // PIC command "finish unloading"
      R     "MAL1S020".PCWrite.ExtFuncOn.FinishCleanSurface; // PIC command "finish unloading"
      R     "MAL1S021".PCWrite.ExtFuncOn.FinishCleanSurface; // PIC command "finish unloading"
      R     "MAL1S022".PCWrite.ExtFuncOn.FinishCleanSurface; // PIC command "finish unloading"
      R     "MAL1S023".PCWrite.ExtFuncOn.FinishCleanSurface; // PIC command "finish unloading"
      R     "MAL1S024".PCWrite.ExtFuncOn.FinishCleanSurface; // PIC command "finish unloading"

//
//MW 2010.04.06      U     "MAL1S032".PCWrite.ExtFuncOn.FinishLoading    // PIC command "finish loading"
//MW 2010.04.06      R     "MAL1S032".PCWrite.ExtFuncOn.FinishLoading    // PIC command "finish loading"
//
      U     "MAL1S032Par".Par.FlagFunction_1.LoadEnd;
      U     "MAL1S032Par".Par.FlagFunction_1.StepLoading; // Step loading
      FP    "MAL1S032Par".Par.FlagFunction_0.ImpulsSollposition;
      =     "MAL1S032Par".Par.FlagFunction_0.MerkerSollpositionFP;
      U     "MAL1S032Par".Par.FlagFunction_0.MerkerSollpositionFP;
      SPBN  fin;
      L     "G266M".A_3111_MXZ41MA.Ma.OutPositionAngle;
      L     "MAL1S032Par".Par.ParIntProcess.LoadingOverlap;
//MW 2010.04.06
      +I    ;
      L     3600; // 360,0°
      >=I   ;
      SPBN  SOZ1;
      -I    ;
      SPA   SOZ2;
SOZ1: NOP   0;
      TAK   ;
SOZ2: NOP   0;
      T     "G266M".A_3111_MXZ41MA.Ma.InPositionTarget;
      SET   ;
//MW 2010.04.06      S     "G266M".TurningTo_Parkposition
      S     "MAL1S032Par".Par.FlagMachine.WEGMESSUNG_0_FLAG;

// Extra Planierrunde wenn der Fahrantrieb ueber 346° beim Beladen Ende war
      L     "G266M".A_3111_MXZ41MA.Ma.OutPositionAngle;
      L     3460; // 346,0 °
      >I    ;
      S     "G266M".Turning_One_Round_More;

// Beladehöhe speichern
      L     "MAL1S032Par".Par.MachineValue.SOLLWERT_HUBZUG1_HOEHE;
      T     "MAL1S032Par".Par.ParIntMachine.LastLoadingLevel; // saved loading value
fin:  NOP   0;

// Hubzüge erst auf der Parkposition abheben
//MW 2010.04.06      U     "G266M".TurningTo_Parkposition
//MW 2010.04.06      FN    "G265M".USW8
//MW 2010.04.06      =     "G265M".USW9

//MW 2010.04.06      U     "G265M".USW9
//MW 2010.04.06      O
//MW 2010.04.06      U     "MAL1S032Par".Par.FlagFunction_1.FinishLoading
//MW 2010.04.06      U(
//MW 2010.04.06      U     "G266M".A_3111_MXZ41MA.A_3111_BZS43.StCtoTrue    // sensor zero point
//MW 2010.04.06      O     "G266M".A_3111_MXZ41MA.A_3111_BZS43.StTrue    // sensor zero point
//MW 2010.04.06      )
//MW 2010.04.06      SPBN  auf
//MW 2010.04.06      L     "G265M".A_3111_MXZ21_31MA.Ma.Par.ParPositionTopLeftUnits    //LIFTING DRIVE
//MW 2010.04.06      L     150
//MW 2010.04.06      +I
//MW 2010.04.06      T     "MAL1S032Par".Par.MachineValue.SOLLWERT_HUBZUG1_HOEHE
//MW 2010.04.06      L     "G265M".A_3111_MXZ21_31MA.Ma.Par.ParPositionTopRightUnits    //LIFTING DRIVE
//MW 2010.04.06      L     150
//MW 2010.04.06      +I
//MW 2010.04.06      T     "MAL1S032Par".Par.MachineValue.SOLLWERT_HUBZUG2_HOEHE
//MW 2010.04.06      L     1
//MW 2010.04.06      T     "G265M".A_3111_MXZ21_31MA.Ma.Par.ParTolPosition
//MW 2010.04.06 auf:  NOP   0
      NOP   0;
NETWORK
TITLE =ASW_6080: Processtime Kilning
//      CALL  "SSA_MH_ProcessTime_Fct" , DB1017
//       InfDataReady :="MAL1S017".ToASW.InfDataReady
//       ProzessActive:="MAL1S017Par".Par.FlagProcess.ProcessActive
//       InStartTime  :="MAL1S017Par".Prozesstime.Starttime
//       OutStartTime :="MAL1S017Par".Prozesstime.Starttime
//       ProcessTime  :="MAL1S017Par".Prozesstime
//
      CALL "SSA_MH_ProcessTime_Fct" , DB  1032 (
           InfDataReady             := "MAL1S032".ToASW.InfDataReady,
           ProzessActive            := "MAL1S032Par".Par.FlagProcess.ProcessActive,
           InStartTime              := "MAL1S032Par".Processtime.StartTime,
           OutStartTime             := "MAL1S032Par".Processtime.StartTime,
           ProcessTime              := "MAL1S032Par".Processtime);

NETWORK
TITLE =Sub 7020: Step start process kilning
//      U     "MAL1S032".ToASW.InfDataReady
//      U     "MAL1S032".PCRead.Step.StActive
////      U     "MAL1S032".PCWrite.ExtFuncOn.StartProcess    // PIC command
//"start
//process kilning"
//      U     "MAL1S032Par".Par.FlagFunction_1.LoadEnd
//
//      U     "G266M".A_3111_MXZ41MA.A_3111_BZS43.StTrue    // sensor zero point
//      U     "G265M".A_3111_MXZ21_31MA.A_3111_BZS23.InpTrue
//      U     "G265M".A_3111_MXZ21_31MA.A_3111_BZS33.InpTrue
//
//      O(
//      UN    "MAL1S032".SecNom.Par1On.Cmd01    // With Loading
//      UN    "MAL1S032".ToASW.InfSameBatchPrevSec
//      U     "MAL1S032".ToASW.InfDataReady
//      U     "MAL1S032".PCRead.Step.StActive
//      )
//
//      S     "MAL1S032Par".Par.FlagFunction_1.FinishLoading    // start process
//kilning
//      R     "MAL1S032Par".Par.FlagFunction_1.LoadEnd
////
//      U     "MAL1S032".PCWrite.ExtFuncOn.StartProcess    // PIC command "start
//process kilning"
//      R     "MAL1S032".PCWrite.ExtFuncOn.StartProcess    // PIC command "start
//process kilning"
////
//      U     "G266M".A_3111_MXZ41MA.Ma.StAdjusted
//      O     "G266M".A_3111_MXZ41MA.Ma.OutAdjusted
//      U     "MAL1S032Par".Par.FlagFunction_1.FinishLoading    // start process
//kilning
//      O     "MAL1S032Par".Par.FlagProcess.ProcessActive
//      SPBN  E702
//      L     "G265M".A_3111_MXZ21_31MA.Ma.Par.ParPositionTopLeftUnits
////LIFTING DRIVE
//      L     50                          //jk
//      +I
//      T     "MAL1S032Par".Par.MachineValue.SOLLWERT_HUBZUG1_HOEHE
//      L     "G265M".A_3111_MXZ21_31MA.Ma.Par.ParPositionTopRightUnits
////LIFTING DRIVE
//      L     50                          //jk
//      +I
//      T     "MAL1S032Par".Par.MachineValue.SOLLWERT_HUBZUG2_HOEHE
//      L     1
//      T     "G265M".A_3111_MXZ21_31MA.Ma.Par.ParTolPosition
//
//E702: NOP   0
//
//      U     "G266M".TurningTo_Parkposition
//      SPBN  E703
//      U(
//      L     "G266M".A_3111_MXZ41MA.Ma.OutPositionAngle
//      L     3500
//      >=I
//      )
//      SPBN  E703
//      L     10                          // 10% speed to parkposition
//      T     "MAL1S032Par".Par.MachineValue.SollwertFahrantrieb
//E703: NOP   0
//
//      U     "G266M".TurningTo_Parkposition
//      SPBN  E704
//      U(
//      L     "G266M".A_3111_MXZ41MA.Ma.OutPositionAngle
//      L     3500
//      <I
//      )
//      SPBN  E704
//      L     87                          // 87% speed to parkposition
//      T     "MAL1S032Par".Par.MachineValue.SollwertFahrantrieb
//E704: NOP   0
//
//MW 2010.04.06
      U     "MAL1S032".ToASW.InfDataReady;
      U     "MAL1S032".PCRead.Step.StActive;
      U     "MAL1S032Par".Par.FlagFunction_1.LoadEnd;
      U     "G266M".A_3111_MXZ41MA.Ma.StAdjusted; // travelling drive on target position
//-Without loading---
      O(    ;
      UN    "MAL1S032".SecNom.Par1On.Cmd01; // With Loading
      UN    "MAL1S032".ToASW.InfSameBatchPrevSec;
      U     "MAL1S032".ToASW.InfDataReady;
      U     "MAL1S032".PCRead.Step.StActive;
      )     ;
      O(    ;
      U     "MAL1S032".PCWrite.ExtFuncOn.FinishLoading; // PIC command "finish loading"
      U     "MAL1S032Par".Par.FlagFunction_1.LoadEnd;
      UN    "MAL1S032".ToASW.InfSameBatchPrevSec;
      U     "MAL1S032".ToASW.InfDataReady;
      U     "MAL1S032".PCRead.Step.StActive;
      )     ;
      S     "MAL1S032Par".Par.FlagFunction_1.FinishLoading; // start process kilning
      R     "MAL1S032Par".Par.FlagFunction_1.LoadEnd;
//MW 2010.04.23
      S     "MAL1S032".PCRead.Status.StaLoaded;
//
      U     "MAL1S032".PCWrite.ExtFuncOn.FinishLoading; // PIC command "finish loading"
      R     "MAL1S032".PCWrite.ExtFuncOn.FinishLoading; // PIC command "finish loading"
//
//-With loading---
      U(    ;
      U     "G266M".A_3111_MXZ41MA.Ma.StAdjusted;
      O     "G266M".A_3111_MXZ41MA.Ma.OutAdjusted;
      U     "MAL1S032Par".Par.FlagFunction_1.FinishLoading; // start process kilning
      )     ;
//-Without loading---
      O(    ;
      UN    "MAL1S032".SecNom.Par1On.Cmd01; // With Loading
      UN    "MAL1S032".ToASW.InfSameBatchPrevSec;
      U     "MAL1S032".PCRead.Step.StReady;
      U     "MAL1S032Par".Par.FlagProcess.ProcessActive;
      )     ;
      O(    ;
      U     "MAL1S032".PCRead.Step.StReady;
      U     "MAL1S032Par".Par.FlagProcess.ProcessActive;
      UN    "MAL1S032Par".Par.FlagFunction_1.StepLoading;
      UN    "MAL1S032Par".Par.FlagFunction_1.FinishLoading;
      UN    "MAL1S032Par".Par.FlagFunction_1.LoadEnd;
      UN    "MAL1S032Par".Par.FlagMachine.WEGMESSUNG_0_FLAG;
      )     ;
      SPB   pPos;
      SPA   E702;
pPos: NOP   0;
      L     "G265M".A_3111_MXZ21_31MA.Ma.Par.ParPositionTopLeftUnits; //LIFTING DRIVE
      L     50;
      +I    ;
      T     "MAL1S032Par".Par.MachineValue.SOLLWERT_HUBZUG1_HOEHE;
      L     "G265M".A_3111_MXZ21_31MA.Ma.Par.ParPositionTopRightUnits; //LIFTING DRIVE
      L     50;
      +I    ;
      T     "MAL1S032Par".Par.MachineValue.SOLLWERT_HUBZUG2_HOEHE;
      L     3;
      T     "G265M".A_3111_MXZ21_31MA.Ma.Par.ParTolPosition;
E702: NOP   0;
NETWORK
TITLE =ASW_8000:  Step unloading kilning
//      UN    "MAL1S032Par".Par.FlagFunction_1.StepUnloading    // Step Unloading
//      R     "MAL1S032Par".Par.FlagFunction_0.OverlapSaved    // Ueberlappung
//erfasst
////
//      U     "MAL1S032".ToASW.InfDataReady
//      U     "MAL1S032".PCRead.Step.StEmptying
//      U(
//      L     "MAL1S032Par".RecipeHeader.Unloading.StartUnloadAuto
////StartUnloadAuto = 0
//      L     1
//      <>I
//      U     "MAL1S032".PCWrite.ExtFuncOn.StartUnLoading    // PIC command
//"start
//unloading"
//      O
//      U(
//      L     "MAL1S032Par".RecipeHeader.Unloading.StartUnloadAuto
////StartUnloadAuto = 10
//      L     1
//      ==I
//      )
//      UN    DB371.DBX  832.1            // 30% Ventilatordrehzahl
//      UN    DB371.DBX 1856.1            // 30% Ventilatordrehzahl
//      )
//      S     "MAL1S032Par".Par.FlagFunction_1.StepUnloading    // Step Unloading
//      R     "MAL1S032Par".Par.FlagMachine.ImpulsNullstellung
//      R     "MAL1S023Par".Par.FlagMachine.WEGMESSUNG_0
//      R     DB922.DBX  148.0            // FP
//      R     "MAL1S032Par".Par.FlagMachine.CmdTurnRevAfterUnloading
//      R     "MAL1S032Par".Par.FlagMachine.CmdTurnFwdAfterUnloading
////
//      SET
//      R     "MAL1S032".PCWrite.ExtFuncOn.StartUnLoading    // PIC command
//"start
//unloading"
////
//      U     "MAL1S032".ToASW.InfDataReady
//      U     "MAL1S032".PCRead.Step.StEmptying
//      U     "MAL1S032Par".Par.FlagFunction_1.StepUnloading    // Step Unloading
//      SPBN  e800
//      L     "MAL1S032Par".Par.ParIntMachine.LastLoadingLevel    // saved
//loading
//value
//      T     "MAL1S032Par".Par.ParIntMachine.FUELLHOEHE_PRODUKT
////
//      U(
//      L     "G265M".A_3111_MXZ21_31MA.Ma.OutPositionLeft
//      L     "MAL1S032Par".Par.ParIntMachine.FUELLHOEHE_PRODUKT
//      >I
//      )
//      O(
//      L     "G265M".A_3111_MXZ21_31MA.Ma.OutPositionRight
//      L     "MAL1S032Par".Par.ParIntMachine.FUELLHOEHE_PRODUKT
//      >I
//      )
//      UN(
//      U(
//      L     "G265M".A_3111_MXZ21_31MA.Ma.OutPositionLeft
//      L     "MAL1S032Par".Par.MachineValue.SOLLWERT_HUBZUG1_HOEHE
//      <=I
//      )
//      U(
//      L     "G265M".A_3111_MXZ21_31MA.Ma.OutPositionRight
//      L     "MAL1S032Par".Par.MachineValue.SOLLWERT_HUBZUG1_HOEHE
//      <=I
//      )
//      )
//      =     "MAL1S032Par".Par.FlagFunction_0.ScrewAboveProductLayer    //
//HubzuegeUeberProdukt
////
////- Letzte Entladehoehe erreicht ---
//      U(
//      L     "MAL1S032Par".Par.MachineValue.SOLLWERT_HUBZUG1_HOEHE
//      L     0
//      <=I
//      )
//      U(
//      L     "MAL1S032Par".Par.MachineValue.SOLLWERT_HUBZUG1_HOEHE
//      L     "G265M".A_3111_MXZ21_31MA.Ma.InPositionTarget
//      ==I
//      )
//      U     "G265M".A_3111_MXZ21_31MA.Ma.StAdjusted
//      U     "MAL1S032Par".Par.FlagFunction_1.StepUnloading    // Step Unloading
//      FP    "MAL1S032Par".Par.FlagFunction_0.UnloadLevelReachedFP    //
//UnloadLevelReachedFP
//      =     "MAL1S032Par".Par.FlagFunction_0.ImpulsUnloadLevelReached    //
//ImpulsUnloadLevelReached
//      UN    "MAL1S032Par".Par.FlagFunction_0.ImpulsUnloadLevelReached    //
//ImpulsUnloadLevelReached
//      O     "MAL1S032Par".Par.FlagFunction_0.OverlapSaved    // Ueberlappung
//erfasst
//      SPB   over
//      L     "G266M".A_3111_MXZ41MA.Ma.OutCntRound
//      L     1
//      +I
//      T     "MAL1S032Par".Par.ParIntProcess.UnloadungRounds
////
//      L     "G266M".A_3111_MXZ41MA.Ma.OutPositionAngle
//      L     3600                        // 360,0°
//      >=I
//      SPBN  soz1
//      -I
//      SPA   soz2
//soz1: NOP   0
//      TAK
//soz2: NOP   0
//      L     100                         // 10,0°
//      +I
//      T     "MAL1S032Par".Par.ParIntProcess.UnloadingOverlap
//      T     "G266M".A_3111_MXZ41MA.Ma.InPositionTarget
//      S     "MAL1S032Par".Par.FlagFunction_0.OverlapSaved    // Ueberlappung
//erfasst
//over: NOP   0
//      U(
//      L     "G266M".A_3111_MXZ41MA.Ma.OutCntRound
//      L     L#0
//      ==D
//      )
//      SPB   rnd1
//      L     "G266M".A_3111_MXZ41MA.Ma.OutCntRound
//      L     L#1
//      ==D
//      SPB   rnd2
//      L     "G266M".A_3111_MXZ41MA.Ma.OutCntRound
//      L     L#2
//      >=D
//      SPB   rnd3
//      SPA   e801
//rnd1: NOP   0
//      L     "MAL1S032Par".RecipeHeader.Unloading.UnLoadingLevelRound_1
//      T     "MAL1S032Par".Par.MachineValue.SOLLWERT_HUBZUG1_HOEHE
//      T     "MAL1S032Par".Par.MachineValue.SOLLWERT_HUBZUG2_HOEHE
//      L     1
//      T     "G265M".A_3111_MXZ21_31MA.Ma.Par.ParTolPosition
//      L     "MAL1S032Par".RecipeHeader.Unloading.UnLoadingSpeed_1
//      T     "MAL1S032Par".Par.MachineValue.SollwertFahrantrieb
//      SPA   e801
//rnd2: NOP   0
//      L     "MAL1S032Par".RecipeHeader.Unloading.UnLoadingLevelRound_2
//      T     "MAL1S032Par".Par.MachineValue.SOLLWERT_HUBZUG1_HOEHE
//      T     "MAL1S032Par".Par.MachineValue.SOLLWERT_HUBZUG2_HOEHE
//      L     1
//      T     "G265M".A_3111_MXZ21_31MA.Ma.Par.ParTolPosition
//      L     "MAL1S032Par".RecipeHeader.Unloading.UnLoadingSpeed_2
//      T     "MAL1S032Par".Par.MachineValue.SollwertFahrantrieb
//      SPA   e801
//rnd3: NOP   0
//      L     "MAL1S032Par".RecipeHeader.Unloading.UnLoadingLevelRound_3
//      T     "MAL1S032Par".Par.MachineValue.SOLLWERT_HUBZUG1_HOEHE
//      T     "MAL1S032Par".Par.MachineValue.SOLLWERT_HUBZUG2_HOEHE
//      L     1
//      T     "G265M".A_3111_MXZ21_31MA.Ma.Par.ParTolPosition
//      L     "MAL1S032Par".RecipeHeader.Unloading.UnLoadingSpeed_3
//      T     "MAL1S032Par".Par.MachineValue.SollwertFahrantrieb
//      SPA   e801
//
//e801: NOP   0
//      U     "MAL1S032".ToASW.InfDataReady
//      U     "MAL1S032".PCRead.Step.StEmptying
//      U     "MAL1S032Par".Par.FlagFunction_1.StepUnloading    // Step Unloading
//      U(
//      L     "G266M".A_3111_MXZ41MA.Ma.OutCntRound
//      L     "MAL1S032Par".Par.ParIntProcess.UnloadungRounds
//      >=I
//      )
//      U     "G265M".A_3111_MXZ21_31MA.Ma.StAdjusted
//      U     "G266M".A_3111_MXZ41MA.Ma.StAdjusted
//      S     "MAL1S032Par".Par.FlagFunction_1.FinishUnloading
//
//      U     "MAL1S032".ToASW.InfDataReady
//      U     "MAL1S032".PCRead.Step.StEmptying
//      U     "MAL1S032Par".Par.FlagFunction_1.FinishUnloading
//      SPBN  e800
//      L     "G265M".A_3111_MXZ21_31MA.Ma.Par.ParPositionTopLeftUnits
//      L     50
//      +I
//      T     "MAL1S032Par".Par.MachineValue.SOLLWERT_HUBZUG1_HOEHE
//      L     "G265M".A_3111_MXZ21_31MA.Ma.Par.ParPositionTopRightUnits
//      L     50
//      +I
//      T     "MAL1S032Par".Par.MachineValue.SOLLWERT_HUBZUG2_HOEHE
//      L     1
//      T     "G265M".A_3111_MXZ21_31MA.Ma.Par.ParTolPosition
//
//      L     0
//      T     "MAL1S032Par".Par.ParIntMachine.LastLoadingLevel    // saved
//loading
//value
//      T     "MAL1S032Par".Par.ParIntMachine.FUELLHOEHE_PRODUKT
//e800: NOP   0
////
//// --> Wie bei der Bank Avangard
//      U     "MAL1S032Par".Par.FlagFunction_1.StepUnloading
//      U     "MAL1S032Par".Par.FlagFunction_1.FinishUnloading
//      FP    DB922.DBX  148.0
//      =     DB922.DBX  148.1
//      SPBN  TAU1
//      L     "G266M".A_3111_MXZ41MA.Ma.OutPositionAngle
//      L     1800
//      <I
//      S     "MAL1S032Par".Par.FlagMachine.CmdTurnRevAfterUnloading
//      L     "G266M".A_3111_MXZ41MA.Ma.OutPositionAngle
//      L     1800
//      >=I
//      S     "MAL1S032Par".Par.FlagMachine.CmdTurnFwdAfterUnloading
//TAU1: NOP   0
//      U     "MAL1S032Par".Par.FlagMachine.CmdTurnRevAfterUnloading
//      O     "MAL1S032Par".Par.FlagMachine.CmdTurnFwdAfterUnloading
//      U     "MAL1S032Par".Par.FlagFunction_1.FinishUnloading
//      U     "G267M".A_3111_MXZ11.StStopped
//      U     "G265M".A_3111_MXZ21_31MA.Ma.OutHigherMinPos
//      U(
//      U     "G265M".A_3111_MXZ21_31MA.A_3111_BZS33.InpTrue
//      U     "G265M".A_3111_MXZ21_31MA.A_3111_BZS23.InpTrue
//      O     "G265M".A_3111_MXZ21_31MA.Ma.StAdjusted
//      )
//      S     "MAL1S032Par".Par.FlagMachine.WEGMESSUNG_0
////
//      U     "MAL1S032".ToASW.InfDataReady
//      U     "MAL1S032Par".Par.FlagFunction_1.FinishUnloading
//      U     "MAL1S032Par".Par.FlagMachine.WEGMESSUNG_0
//      SPBN  TAU2
////    L     "MAL1S032Par".RecipeHeader.Cleaning.CleaningSpeed_1
//      L     30                          // 30%
//      T     "MAL1S032Par".Par.MachineValue.SollwertFahrantrieb
//TAU2: NOP   0
//      NOP   0
//
//MW 2010.04.06
      UN    "MAL1S032Par".Par.FlagFunction_1.StepUnloading; // Step Unloading
      R     "MAL1S032Par".Par.FlagFunction_0.OverlapSaved; // Ueberlappung erfasst
//
      U     "MAL1S032".ToASW.InfDataReady;
      U     "MAL1S032".PCRead.Step.StEmptying;
      U(    ;
      L     "MAL1S032Par".RecipeHeader.Unloading.StartUnloadAuto; //StartUnloadAuto = 0
      L     1;
      <>I   ;
      U     "MAL1S032".PCWrite.ExtFuncOn.StartUnLoading; // PIC command "start unloading"
      O     ;
      U(    ;
      L     "MAL1S032Par".RecipeHeader.Unloading.StartUnloadAuto; //StartUnloadAuto = 10
      L     1;
      ==I   ;
      )     ;
      UN    "G271M".A_3125_TSC01_AF.OutL; // 30% Ventilatordrehzahl
      UN    "G271M".A_3126_TSC01_AF.OutL; // 30% Ventilatordrehzahl
      )     ;
      S     "MAL1S032Par".Par.FlagFunction_1.StepUnloading; // Step Unloading
      R     "MAL1S032Par".Par.FlagMachine.ImpulsNullstellung;
      R     "MAL1S023Par".Par.FlagMachine.WEGMESSUNG_0;
      R     DB922.DBX  148.0; // FP
      R     "MAL1S032Par".Par.FlagMachine.CmdTurnRevAfterUnloading;
      R     "MAL1S032Par".Par.FlagMachine.CmdTurnFwdAfterUnloading;
//
      SET   ;
      R     "MAL1S032".PCWrite.ExtFuncOn.StartUnLoading; // PIC command "start unloading"
//
      U     "MAL1S032".ToASW.InfDataReady;
      U     "MAL1S032".PCRead.Step.StEmptying;
      U     "MAL1S032Par".Par.FlagFunction_1.StepUnloading; // Step Unloading
      SPBN  e800;
//-Start process without loading---
      L     "MAL1S032Par".Par.ParIntMachine.LastLoadingLevel; // saved loading value
      L     0;
      ==I   ;
      L     "MAL1S032Par".RecipeHeader.Loading.LoadingLevelRound_3;
      SPB   LLL;
//-Start process with loading---
      L     "MAL1S032Par".Par.ParIntMachine.LastLoadingLevel; // saved loading value
LLL:  T     "MAL1S032Par".Par.ParIntMachine.FUELLHOEHE_PRODUKT;
//
      U(    ;
      L     "G265M".A_3111_MXZ21_31MA.Ma.OutPositionLeft;
      L     "MAL1S032Par".Par.ParIntMachine.FUELLHOEHE_PRODUKT;
      >I    ;
      )     ;
      O(    ;
      L     "G265M".A_3111_MXZ21_31MA.Ma.OutPositionRight;
      L     "MAL1S032Par".Par.ParIntMachine.FUELLHOEHE_PRODUKT;
      >I    ;
      )     ;
      UN(   ;
      U(    ;
      L     "G265M".A_3111_MXZ21_31MA.Ma.OutPositionLeft;
      L     "MAL1S032Par".Par.MachineValue.SOLLWERT_HUBZUG1_HOEHE;
      <=I   ;
      )     ;
      U(    ;
      L     "G265M".A_3111_MXZ21_31MA.Ma.OutPositionRight;
      L     "MAL1S032Par".Par.MachineValue.SOLLWERT_HUBZUG1_HOEHE;
      <=I   ;
      )     ;
      )     ;
      =     "MAL1S032Par".Par.FlagFunction_0.ScrewAboveProductLayer; // HubzuegeUeberProdukt
//
//- Letzte Entladehoehe erreicht ---
      U(    ;
      L     "MAL1S032Par".Par.MachineValue.SOLLWERT_HUBZUG1_HOEHE;
      L     0;
      <=I   ;
      )     ;
      U(    ;
      L     "MAL1S032Par".Par.MachineValue.SOLLWERT_HUBZUG1_HOEHE;
      L     "G265M".A_3111_MXZ21_31MA.Ma.InPositionTarget;
      ==I   ;
      )     ;
      U     "G265M".A_3111_MXZ21_31MA.Ma.StAdjusted;
      U     "MAL1S032Par".Par.FlagFunction_1.StepUnloading; // Step Unloading
      FP    "MAL1S032Par".Par.FlagFunction_0.UnloadLevelReachedFP; // UnloadLevelReachedFP
      =     "MAL1S032Par".Par.FlagFunction_0.ImpulsUnloadLevelReached; // ImpulsUnloadLevelReached
      UN    "MAL1S032Par".Par.FlagFunction_0.ImpulsUnloadLevelReached; // ImpulsUnloadLevelReached
      O     "MAL1S032Par".Par.FlagFunction_0.OverlapSaved; // Ueberlappung erfasst
      SPB   over;
      L     "G266M".A_3111_MXZ41MA.Ma.OutCntRound;
      L     1;
      +I    ;
      T     "MAL1S032Par".Par.ParIntProcess.UnloadungRounds;
//
      L     "G266M".A_3111_MXZ41MA.Ma.OutPositionAngle;
      L     3600; // 360,0°
      >=I   ;
      SPBN  soz1;
      -I    ;
      SPA   soz2;
soz1: NOP   0;
      TAK   ;
soz2: NOP   0;
//BRT20101018 ====> Overlapping nur noch 5°!!!
//      L     100                         // 10,0°
      L     50; // 5,0°
//<==== BRT20101018
      +I    ;
      T     "MAL1S032Par".Par.ParIntProcess.UnloadingOverlap;
      T     "G266M".A_3111_MXZ41MA.Ma.InPositionTarget;
      S     "MAL1S032Par".Par.FlagFunction_0.OverlapSaved; // Ueberlappung erfasst
over: NOP   0;
      L     "MAL1S032Par".RecipeHeader.Unloading.UnLoadingSpeed_2; //JV290710
      T     "MAL1S032Par".RecipeHeader.Unloading.UnLoadingSpeed_3; //JV290710
//-Only ONE unloading round---  //MW 2010.04.06
// 2 unloading rounds JV290710
//      SPA   rnd1
      U(    ;
      L     "G266M".A_3111_MXZ41MA.Ma.OutCntRound;
      L     L#0;
      ==D   ;
      )     ;
      SPB   rnd1;
      L     "G266M".A_3111_MXZ41MA.Ma.OutCntRound;
      L     L#1;
      ==D   ;
      SPB   rnd2;
      L     "G266M".A_3111_MXZ41MA.Ma.OutCntRound;
      L     L#2;
      >=D   ;
      SPB   rnd3;
      SPA   e801;
rnd1: NOP   0;
      L     "MAL1S032Par".RecipeHeader.Unloading.UnLoadingLevelRound_1;
      T     "MAL1S032Par".Par.MachineValue.SOLLWERT_HUBZUG1_HOEHE;
      T     "MAL1S032Par".Par.MachineValue.SOLLWERT_HUBZUG2_HOEHE;
      L     1;
      T     "G265M".A_3111_MXZ21_31MA.Ma.Par.ParTolPosition;
      L     "MAL1S032Par".RecipeHeader.Unloading.UnLoadingSpeed_1;
      T     "MAL1S032Par".Par.MachineValue.SollwertFahrantrieb;
      SPA   e801;
rnd2: NOP   0;
//JV290710      L     "MAL1S032Par".RecipeHeader.Unloading.UnLoadingLevelRound_2
      L     0; //JV290710   last unloading round
      T     "MAL1S032Par".Par.MachineValue.SOLLWERT_HUBZUG1_HOEHE;
      T     "MAL1S032Par".Par.MachineValue.SOLLWERT_HUBZUG2_HOEHE;
//JV290710      L     1
      L     0;
      T     "G265M".A_3111_MXZ21_31MA.Ma.Par.ParTolPosition;
      L     "MAL1S032Par".RecipeHeader.Unloading.UnLoadingSpeed_2;
      T     "MAL1S032Par".Par.MachineValue.SollwertFahrantrieb;
      SPA   e801;
rnd3: NOP   0;
      L     "MAL1S032Par".RecipeHeader.Unloading.UnLoadingLevelRound_3;
      T     "MAL1S032Par".Par.MachineValue.SOLLWERT_HUBZUG1_HOEHE;
      T     "MAL1S032Par".Par.MachineValue.SOLLWERT_HUBZUG2_HOEHE;
      L     1;
      T     "G265M".A_3111_MXZ21_31MA.Ma.Par.ParTolPosition;
      L     "MAL1S032Par".RecipeHeader.Unloading.UnLoadingSpeed_3;
      T     "MAL1S032Par".Par.MachineValue.SollwertFahrantrieb;
      SPA   e801;

e801: NOP   0;
      U     "MAL1S032".ToASW.InfDataReady;
      U     "MAL1S032".PCRead.Step.StEmptying;
      U     "MAL1S032Par".Par.FlagFunction_1.StepUnloading; // Step Unloading
      U(    ;
      L     "G266M".A_3111_MXZ41MA.Ma.OutCntRound;
      L     "MAL1S032Par".Par.ParIntProcess.UnloadungRounds;
      >=I   ;
      )     ;
      U     "G265M".A_3111_MXZ21_31MA.Ma.StAdjusted;
      U     "G266M".A_3111_MXZ41MA.Ma.StAdjusted;
      S     "MAL1S032Par".Par.FlagFunction_1.FinishUnloading;
//MW 2010.04.06
      R     "MAL1S032Par".Par.FlagProcess.Product_Inside;

      U     "MAL1S032".ToASW.InfDataReady;
      U     "MAL1S032".PCRead.Step.StEmptying;
      U     "MAL1S032Par".Par.FlagFunction_1.FinishUnloading;
      SPBN  e800;
      L     "G265M".A_3111_MXZ21_31MA.Ma.Par.ParPositionTopLeftUnits;
      L     50;
      +I    ;
      T     "MAL1S032Par".Par.MachineValue.SOLLWERT_HUBZUG1_HOEHE;
      L     "G265M".A_3111_MXZ21_31MA.Ma.Par.ParPositionTopRightUnits;
      L     50;
      +I    ;
      T     "MAL1S032Par".Par.MachineValue.SOLLWERT_HUBZUG2_HOEHE;
      L     1;
      T     "G265M".A_3111_MXZ21_31MA.Ma.Par.ParTolPosition;

//MW 2010.04.06      L     0
//MW 2010.04.06      T     "MAL1S032Par".Par.ParIntMachine.LastLoadingLevel    // saved loading value
//MW 2010.04.06      T     "MAL1S032Par".Par.ParIntMachine.FUELLHOEHE_PRODUKT
e800: NOP   0;
//
// --> Wie bei der Bank Avangard
      U     "MAL1S032Par".Par.FlagFunction_1.StepUnloading;
      U     "MAL1S032Par".Par.FlagFunction_1.FinishUnloading;
      FP    DB922.DBX  148.0;
      =     DB922.DBX  148.1;
      SPBN  TAU1;
      L     "G266M".A_3111_MXZ41MA.Ma.OutPositionAngle;
      L     1800;
      <I    ;
      S     "MAL1S032Par".Par.FlagMachine.CmdTurnRevAfterUnloading;
      L     "G266M".A_3111_MXZ41MA.Ma.OutPositionAngle;
      L     1800;
      >=I   ;
      S     "MAL1S032Par".Par.FlagMachine.CmdTurnFwdAfterUnloading;
TAU1: NOP   0;
      U     "MAL1S032Par".Par.FlagMachine.CmdTurnRevAfterUnloading;
      O     "MAL1S032Par".Par.FlagMachine.CmdTurnFwdAfterUnloading;
      U     "MAL1S032Par".Par.FlagFunction_1.FinishUnloading;
      U     "G267M".A_3111_MXZ11.StStopped;
      U     "G265M".A_3111_MXZ21_31MA.Ma.OutHigherMinPos;
      U(    ;
      U     "G265M".A_3111_MXZ21_31MA.A_3111_BZS33.InpTrue;
      U     "G265M".A_3111_MXZ21_31MA.A_3111_BZS23.InpTrue;
      O     "G265M".A_3111_MXZ21_31MA.Ma.StAdjusted;
      )     ;
      S     "MAL1S032Par".Par.FlagMachine.WEGMESSUNG_0;
//
      U     "MAL1S032".ToASW.InfDataReady;
      U     "MAL1S032Par".Par.FlagFunction_1.FinishUnloading;
      U     "MAL1S032Par".Par.FlagMachine.WEGMESSUNG_0;
      SPBN  TAU2;
//    L     "MAL1S032Par".RecipeHeader.Cleaning.CleaningSpeed_1
      L     30; // 30%
      T     "MAL1S032Par".Par.MachineValue.SollwertFahrantrieb;
TAU2: NOP   0;
      NOP   0;
NETWORK
TITLE =ASW_9000: Step cleaning
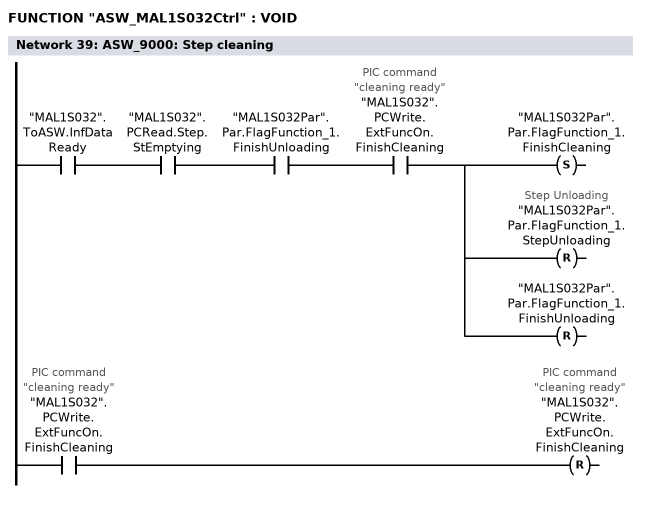

      U     "MAL1S032".ToASW.InfDataReady;
      U     "MAL1S032".PCRead.Step.StEmptying;
      U     "MAL1S032Par".Par.FlagFunction_1.FinishUnloading;
      U     "MAL1S032".PCWrite.ExtFuncOn.FinishCleaning; // PIC command "cleaning ready"
      S     "MAL1S032Par".Par.FlagFunction_1.FinishCleaning;
      R     "MAL1S032Par".Par.FlagFunction_1.StepUnloading; // Step Unloading
      R     "MAL1S032Par".Par.FlagFunction_1.FinishUnloading;
//
      U     "MAL1S032".PCWrite.ExtFuncOn.FinishCleaning; // PIC command "cleaning ready"
      R     "MAL1S032".PCWrite.ExtFuncOn.FinishCleaning; // PIC command "cleaning ready"
NETWORK
TITLE =ASW_9080: Send section date to PIC after germination

      AUF   "MAL1S032";
      U     "MAL1S032".PCRead.Step.StEmptying;
      FP    "MAL1S032Par".Par.FlagProcess.FP_SendResultToPIC;
      SPBN  E908;
//

E908: NOP   0;
NETWORK
TITLE =ASW_9099: Init Flag
////MW 2010.04.06
//-Extended section commands---
      L     0;
      T     #tmpInt;
      CALL "SIEMENS_FILL" (
           BVAL                     := #tmpInt,
           RET_VAL                  := #tmpRET,
           BLK                      := "MAL1S032".PCWrite.ExtFuncOn);

      CALL "SIEMENS_FILL" (
           BVAL                     := #tmpInt,
           RET_VAL                  := #tmpRET,
           BLK                      := "MAL1S032".PCWrite.ExtFuncOff);

NETWORK
TITLE =ASW_10000: ILO functions

      U     "MAL1S032".SecAc.Sta1On.Inf08;
      =     "MAL1S032".Gr.All.Spare04;

//- Little help for PIC-People, Number 3
      UN    "G265M".Gr.InManual; // LIFTING DEVICE KILN 1
      UN    "G266M".Gr.InManual; // TRAVELLING DRIVE KILN 1
      UN    "G267M".Gr.InManual; // UNLOADING / LOADING SCREW KILN 1
      UN    "G268M".Gr.InManual; // DISCHARGE DOOR KILN 1
      UN    "G271M".Gr.InManual; // FAN KILN 1
      UN    "G272M".Gr.InManual; // FRESH AIR LOUVER KILN 1
      UN    "G273M".Gr.InManual; // RECYCLING AIR LOUVER KILN 1
      UN    "G274M".Gr.InManual; // EXHAUST AIR LOUVER KILN 1
      UN    "G276M".Gr.InManual; // HEATING KILN 1
      UN    "G277M".Gr.InManual; // LOUVER AIR HEATER 1 FOR KILN 1
      UN    "G278M".Gr.InManual; // WITHERING AIR KILN 1
      UN    "G279M".Gr.InManual; // HEATING KILN 1 + 2
      FP    DB922.DBX 3029.0;
      =     DB922.DBX 3029.1;
      U     DB922.DBX 3029.1;
      SPBN  RSM3;
      L     0;
      T     "MAL1S032Par".Ilo.Code_ILO_Funktion0; // FCM 32 LINE 1 SEC 32 KILN
      T     "MAL1S032Par".Ilo.ILOMode;
RSM3: NOP   0;

//- Combination OLD and NEW ---
      U     "MAL1S032".SecAc.Sta1On.Inf08;
      SPBN  IFM;
      L     "MAL1S032Par".Ilo.ILOMode;
      L     100;
      *I    ;
      T     "MAL1S032Par".Ilo.Code_ILO_Funktion0;
IFM:  NOP   0;

//  no ILO-mode >> cmd manual off to all used groups and reset all flags
      U     "MAL1S032".SecAc.Sta1On.Inf08;
      FN    "MAL1S032Par".Ilo.Flag.EdgeILOModeOn;
//MW 2010.04.06      S     "MAL1S032Par".Ilo.GrCMDManOff[1]    // (ManOff)
//MW 2010.04.06      R     "MAL1S032Par".Ilo.GrCMDManAdditional.Cmd1[1]
//MW 2010.04.06      R     "MAL1S032Par".Ilo.GrCMDManAdditional.Cmd2[2]
//  Gr-cmd manual OFF
      S     "G265M".Gr.CmdManualOff; // LIFTING DEVICE KILN 1
      S     "G266M".Gr.CmdManualOff; // TRAVELLING DRIVE KILN 1
      S     "G267M".Gr.CmdManualOff; // UNLOADING / LOADING SCREW KILN 1
      S     "G268M".Gr.CmdManualOff; // DISCHARGE DOOR KILN 1
      S     "G271M".Gr.CmdManualOff; // FAN KILN 1
      S     "G272M".Gr.CmdManualOff; // FRESH AIR LOUVER KILN 1
      S     "G273M".Gr.CmdManualOff; // RECYCLING AIR LOUVER KILN 1
      S     "G274M".Gr.CmdManualOff; // EXHAUST AIR LOUVER KILN 1
      S     "G276M".Gr.CmdManualOff; // HEATING KILN 1
      S     "G277M".Gr.CmdManualOff; // LOUVER AIR HEATER 1 FOR KILN 1
      S     "G278M".Gr.CmdManualOff; // WITHERING AIR KILN 1
      S     "G279M".Gr.CmdManualOff; // HEATING KILN 1 + 2
//  RESET ADDITIONAL CMD`S
      R     "G265M".USW14; // ILO-cmd
      R     "G265M".USW15; // ILO-cmd
      R     "G266M".USW14; // ILO-cmd
      R     "G266M".USW15; // ILO-cmd
      R     "G267M".USW14; // ILO-cmd
      R     "G267M".USW15; // ILO-cmd
      R     "G268M".USW14; // ILO-cmd
      R     "G268M".USW15; // ILO-cmd
      R     "G271M".USW14; // ILO-cmd
      R     "G271M".USW15; // ILO-cmd
      R     "G272M".USW14; // ILO-cmd
      R     "G272M".USW15; // ILO-cmd
      R     "G273M".USW14; // ILO-cmd
      R     "G273M".USW15; // ILO-cmd
      R     "G274M".USW14; // ILO-cmd
      R     "G274M".USW15; // ILO-cmd
      R     "G276M".USW14; // ILO-cmd
      R     "G276M".USW15; // ILO-cmd
      R     "G277M".USW14; // ILO-cmd
      R     "G277M".USW15; // ILO-cmd
      R     "G278M".USW14; // ILO-cmd
      R     "G278M".USW15; // ILO-cmd
      R     "G279M".USW14; // ILO-cmd
      R     "G279M".USW15; // ILO-cmd

//MW 2010.04.06
//- Little help for PIC-People, Number 2
      U     "MAL1S032".SecAc.Sta1On.Inf08;
      SPB   RSM2;
      L     0;
      T     #tmpInt;
      CALL "SIEMENS_FILL" (
           BVAL                     := #tmpInt,
           RET_VAL                  := #tmpRET,
           BLK                      := "MAL1S032Par".Ilo);
RSM2: NOP   0;

